// TwinCAT 3 PLC project Untitled1
// ProgramVersion: 3.1.4023.0
// libraries:
//   Tc2_SerialCom, * (Beckhoff Automation GmbH)
//   Tc2_Standard, * (Beckhoff Automation GmbH)
//   Tc2_System, * (Beckhoff Automation GmbH)
//   Tc2_Utilities, * (Beckhoff Automation GmbH)
//   Tc3_Database, * (Beckhoff Automation GmbH)
//   Tc3_IotBase, * (Beckhoff Automation GmbH)
//   Tc3_Module, * (Beckhoff Automation GmbH)
// project tree:
//   DUTs/ ST_SelectStructData.TcDUT, ST_SelectStructIMU.TcDUT
//   GVLs/ GVL.TcGVL
//   / PlcTask_Background.TcTTO, PlcTask_Buffer.TcTTO, PlcTask_Send.TcTTO, PlcTask_Read.TcTTO, PlcTask_Vacuum.TcTTO (not stored)
//   POUs/ Background_FatigueCam.TcPOU, Background_GPS.TcPOU, Background_IMU.TcPOU, Background_Time.TcPOU (not stored), Buffer_Data.TcPOU, Buffer_IMU.TcPOU, FB_FatigueCam_Receive.TcPOU (not stored), Get_Data.TcPOU, Get_IMU.TcPOU, Main_Background.TcPOU, Main_Read.TcPOU, Main_SendIMU.TcPOU, Main_Send.TcPOU, Main_Vacuum.TcPOU, Read_IMU.TcPOU, Read_Pressure.TcPOU, Read_Payload.TcPOU, Main_Buffer.TcPOU, Main_SendData.TcPOU, Read_FatigueCam.TcPOU, Read_GPS.TcPOU, Read_ID.TcPOU, Save_Data.TcPOU, Save_IMU.TcPOU, Send_Data.TcPOU, Send_IMU.TcPOU, Vacuum_Buffer_Data.TcPOU, Vacuum_Buffer_Data_2.TcPOU (not stored), Vacuum_Buffer_IMU.TcPOU, Vacuum_Buffer_IMU_2.TcPOU, Vacuum_Data.TcPOU, Vacuum_IMU.TcPOU
// real-time tasks:
//   TASK PlcTask_Buffer: cycle T#2333.1us, priority 20, ADS port 351
//   TASK PlcTask_Read: cycle T#999.9us, priority 19, ADS port 350
//   TASK PlcTask_Send: cycle T#4332.9us, priority 21, ADS port 352
//   TASK PlcTask_Background: cycle T#333.3us, priority 18, ADS port 349
//   TASK PlcTask_Vacuum: cycle T#333.3us, priority 16, ADS port 348
// I/O:
//   DEVICE Device 1 (EtherCAT) (disabled), AmsNetId 5.95.29.222.2.1
//     Term 1 (EK1200) [EK1200-5000 EtherCAT Power supply (2A E-Bus)]
//       Term 2 (EL9221-5000) [EL9221-5000 Overcurrent protection 24V DC, 1Ch., max. 10A, adjustable]
//       Term 3 (EL9011) [EL9011 End Terminal]
//   DEVICE Device 4 (EtherCAT) (disabled), AmsNetId 5.95.29.222.5.1
//     Term 4 (EK1101) [EK1101 EtherCAT Coupler (2A E-Bus, ID switch)]
//       Term 5 (EL9221-5000) [EL9221-5000 Overcurrent protection 24V DC, 1Ch., max. 10A, adjustable]
//       Term 6 (EL3052) [EL3052 2Ch. Ana. Input 4-20mA]
//       Term 7 (EL3061) [EL3061 1Ch. Ana. Input 0-10V]
//       Term 8 (EL6001) [EL6001 Interface (RS232)]
//       Term 9 (EL9505) [EL9505 Power supply terminal 5V]
//       Term 13 (EL9011) [EL9011 End Terminal]
//     Term 10 (EK1101) [EK1101 EtherCAT Coupler (2A E-Bus, ID switch)]
//       Term 11 (EL9221-5000) [EL9221-5000 Overcurrent protection 24V DC, 1Ch., max. 10A, adjustable]
//       Term 12 (EL3052) [EL3052 2Ch. Ana. Input 4-20mA]
//       Term 13 (EL3061) [EL3061 1Ch. Ana. Input 0-10V]
//       Term 14 (EL6001) [EL6001 Interface (RS232)]
//       Term 15 (EL9505) [EL9505 Power supply terminal 5V]
//       Term 14 (EL9011) [EL9011 End Terminal]
//   DEVICE Device 3 (COM Port) (disabled)
// variable links:
//   Untitled1/Untitled1 Instance <-> Device 4 (EtherCAT)/Term 10 (EK1101)
//     PlcTask_Read Inputs/GVL.Rear_Trailer_State <-> InfoData/State
//     PlcTask_Read Inputs/Read_ID.Trailer_ID_Rear <-> ID/ID
//   Untitled1/Untitled1 Instance <-> Device 4 (EtherCAT)/Term 10 (EK1101)/Term 12 (EL3052)
//     PlcTask_Read Inputs/Read_Pressure.EL3052_Rear_Bit <-> AI Standard Channel 1/Value
//   Untitled1/Untitled1 Instance <-> Device 4 (EtherCAT)/Term 10 (EK1101)/Term 13 (EL3061)
//     PlcTask_Read Inputs/Read_Payload.EL3061_Rear_Bit <-> AI Standard/Value
//   Untitled1/Untitled1 Instance <-> Device 4 (EtherCAT)/Term 10 (EK1101)/Term 14 (EL6001)
//     PlcTask_Send Inputs/Background_IMU.stIn_EL6001_Rear/D[{0..21}] <-> COM Inputs/Data In {0..21}  (22 links)
//     PlcTask_Send Inputs/Background_IMU.stIn_EL6001_Rear/Status <-> COM Inputs/Status
//     PlcTask_Send Outputs/Background_IMU.stOut_EL6001_Rear/Ctrl <-> COM Outputs/Ctrl
//     PlcTask_Send Outputs/Background_IMU.stOut_EL6001_Rear/D[{0..21}] <-> COM Outputs/Data Out {0..21}  (22 links)
//   Untitled1/Untitled1 Instance <-> Device 4 (EtherCAT)/Term 4 (EK1101)
//     PlcTask_Read Inputs/GVL.Lead_Trailer_State <-> InfoData/State
//     PlcTask_Read Inputs/Read_ID.Trailer_ID_Lead <-> ID/ID
//   Untitled1/Untitled1 Instance <-> Device 4 (EtherCAT)/Term 4 (EK1101)/Term 6 (EL3052)
//     PlcTask_Read Inputs/Read_Pressure.EL3052_Lead_Bit <-> AI Standard Channel 1/Value
//   Untitled1/Untitled1 Instance <-> Device 4 (EtherCAT)/Term 4 (EK1101)/Term 7 (EL3061)
//     PlcTask_Read Inputs/Read_Payload.EL3061_Lead_Bit <-> AI Standard/Value
//   Untitled1/Untitled1 Instance <-> Device 4 (EtherCAT)/Term 4 (EK1101)/Term 8 (EL6001)
//     PlcTask_Send Inputs/Background_IMU.stIn_EL6001_Lead/D[{0..21}] <-> COM Inputs/Data In {0..21}  (22 links)
//     PlcTask_Send Inputs/Background_IMU.stIn_EL6001_Lead/Status <-> COM Inputs/Status
//     PlcTask_Send Outputs/Background_IMU.stOut_EL6001_Lead/Ctrl <-> COM Outputs/Ctrl
//     PlcTask_Send Outputs/Background_IMU.stOut_EL6001_Lead/D[{0..21}] <-> COM Outputs/Data Out {0..21}  (22 links)

CONFIGURATION Untitled1
    RESOURCE PLC ON TwinCAT3
        TASK PlcTask_Background(INTERVAL := ?, PRIORITY := 18);
        TASK PlcTask_Buffer(INTERVAL := T#2333.1us, PRIORITY := 20);
        TASK PlcTask_Send(INTERVAL := T#97323.6us, PRIORITY := 21);
        TASK PlcTask_Read(INTERVAL := T#999.9us, PRIORITY := 19);
        PROGRAM Main_Background WITH PlcTask_Background : Main_Background;
        PROGRAM Main_Buffer WITH PlcTask_Buffer : Main_Buffer;
        PROGRAM Main_Send WITH PlcTask_Send : Main_Send;
        PROGRAM Main_Read WITH PlcTask_Read : Main_Read;
    END_RESOURCE
END_CONFIGURATION

// ---- DUTs/ST_SelectStructData.TcDUT
TYPE ST_SelectStructData :
STRUCT
	TimeStr			: DATE_AND_TIME;	
	Trailer_ID		: UINT;
	Lat				: LREAL;
	Lon				: LREAL;
	Speed			: LREAL;
	Overspeed		: BOOL;
	Payload_EMA		: LREAL;
	Payload_Raw		: LREAL;
	Overload		: BOOL;
	Pressure_Cyl	: LREAL;
	Pressure_Val	: LREAL;
	Strain_Left		: LREAL;
	Strain_Right	: LREAL;
	EventCode		: UINT;
	Cycle_Duration	: UDINT;
	Hyd_Efficiency	: LREAL;
END_STRUCT
END_TYPE

// ---- DUTs/ST_SelectStructIMU.TcDUT
TYPE ST_SelectStructIMU :
STRUCT
	TimeStr			: DATE_AND_TIME;
	Millis			: UINT;	
	Trailer_ID		: UINT;
	RoadSec			: UINT;
	AccX			: LREAL;
	AccY			: LREAL;
	AccZ			: LREAL;
	Pitch			: LREAL;
	Roll			: LREAL;
END_STRUCT
END_TYPE

// ---- GVLs/GVL.TcGVL
{attribute 'qualified_only'}
VAR_GLOBAL
	Lead_Trailer_State AT %I*	: UINT;
	Rear_Trailer_State AT %I*	: UINT;
END_VAR

// ---- POUs/Main_Background.TcPOU
PROGRAM Main_Background
VAR
END_VAR

(* execute background processes *)
Background_Time();
//Background_IMU();
//Background_FatigueCam();
Background_GPS();

END_PROGRAM

// ---- POUs/Background_GPS.TcPOU
PROGRAM Background_GPS

VAR
	RxBuffer	:ComBuffer;
	TxBuffer	:ComBuffer;
	
	fbLineCtrlAds	: SerialLineControlADS;
	bAdsError		: BOOL;
	nAdsErrorID		: UDINT;
	bConnect		: BOOL := TRUE;
	sNetID			: T_amsNetId;
	stSerialCfg		: ComSerialConfig;
	Port			: BOOL;
END_VAR

stSerialCfg.Baudrate := 4800;
stSerialCfg.ComPort := 3;
stSerialCfg.DataBits := 8;
stSerialCfg.Parity := PARITY_NONE;
stSerialCfg.StopBits := STOPBITS_ONE;

fbLineCtrlAds(
	Connect 	:= bConnect,
	SerialCfg	:= stSerialCfg,
	NetId		:= sNetId,
	Timeout		:= T#5s,
	TxBuffer	:= TxBuffer,
	RxBuffer	:= RxBuffer,
	Busy		:= ,
	Error		=> bAdsError,
	ErrorID		=> nAdsErrorID,
	PortOpened	=> Port
);

END_PROGRAM

// ---- POUs/Main_Buffer.TcPOU
PROGRAM Main_Buffer
VAR
	
END_VAR

(* save data to database *)
//Buffer_Data();
Buffer_IMU();

END_PROGRAM

// ---- POUs/Buffer_IMU.TcPOU
PROGRAM Buffer_IMU
VAR
	pSec		: WORD;
	diff		: BOOL;
	
	TimeStr		: ARRAY [1..50] OF STRING;
	//Millis		: ARRAY [1..50] OF STRING;
	Trailer_ID_Lead	: ARRAY [1..50] OF STRING;
	//RoadSec		: ARRAY [1..50] OF STRING;
	Pitch_Lead		: ARRAY [1..50] OF STRING;
	Roll_Lead		: ARRAY [1..50] OF STRING;
	AccX_Lead		: ARRAY [1..50] OF STRING;
	AccY_Lead		: ARRAY [1..50] OF STRING;
	AccZ_Lead		: ARRAY [1..50] OF STRING;
	
	Trailer_ID_Rear	: ARRAY [1..50] OF STRING;
	//RoadSec		: ARRAY [1..50] OF STRING;
	Pitch_Rear		: ARRAY [1..50] OF STRING;
	Roll_Rear		: ARRAY [1..50] OF STRING;
	AccX_Rear		: ARRAY [1..50] OF STRING;
	AccY_Rear		: ARRAY [1..50] OF STRING;
	AccZ_Rear		: ARRAY [1..50] OF STRING;
	
	fbSqlDatabase	: FB_SQLDatabaseEvt(sNetID := '', tTimeout := T#1000S);
	fbSqlCommand	: FB_SQLCommandEvt(sNetID := '', tTimeout := T#1000S);
	fbSqlResult		: FB_SQLResultEvt(sNetID:='', tTimeout   := T#1000S); 
	sCmd			: STRING(500000);
	sCmd2			: STRING(500000);
	nState			: INT;
	nState_Switch	: INT;
	
	aReadStruct		: ST_SelectStructIMU;
	aReadStruct_2	: ST_SelectStructIMU;
	Timestamp		: DT;
	Timestamp_2		: DT; 
	
	Initialized		: BOOL := FALSE;
	Done			: BOOL;
	i				: INT;
	Pragma_Done		: BOOL;
	Counter			: ULINT;
	
	Dbid			: UDINT;
	
	bDisconnect		: BOOL;
END_VAR

(* convert to strings *)
//PrimeMover_ID		:= Read_ID.PrimeMover_ID;
TimeStr				:= Read_IMU.TimeStr;
//Millis			:= Read_IMU.Millis;
Trailer_ID_Lead		:= Read_IMU.Trailer_ID_Lead;
Pitch_Lead			:= Read_IMU.Pitch_Lead;
Roll_Lead			:= Read_IMU.Roll_Lead;
AccX_Lead			:= Read_IMU.AccX_Lead;
AccY_Lead			:= Read_IMU.AccY_Lead;
AccZ_Lead			:= Read_IMU.AccZ_Lead;

Trailer_ID_Rear		:= Read_IMU.Trailer_ID_Rear;
Pitch_Rear			:= Read_IMU.Pitch_Rear;
Roll_Rear			:= Read_IMU.Roll_Rear;
AccX_Rear			:= Read_IMU.AccX_Rear;
AccY_Rear			:= Read_IMU.AccY_Rear;
AccZ_Rear			:= Read_IMU.AccZ_Rear;

IF NOT Initialized THEN
	
	//initialization (choose which database for buffer)
	CASE nState OF
				
		0:
			(* connect to buffer_imu *)	
			IF Vacuum_Buffer_IMU.Vacuumed THEN
				
				Dbid := 2;		
				IF fbSqlDatabase.Connect(Dbid) THEN
					IF fbSqlDatabase.bError THEN
						nState := 255; 
					ELSE
						nState := nState+1;
					END_IF
				END_IF
				
			END_IF
			
			
		1:
			IF fbSqlDatabase.CreateCmd(ADR(fbSqlCommand)) THEN
				IF fbSqlDatabase.bError THEN
					nState := 255; 
				ELSE
					nState := nState+1; 
				END_IF
			END_IF
			
		2:	(* execute pragmas *)
			sCmd	:= 'PRAGMA journal_mode = WAL; PRAGMA synchronous = NORMAL; PRAGMA temp_store = MEMORY; PRAGMA mmap_size = 30000000000; PRAGMA page_size = 32768; PRAGMA locking_mode = EXCLUSIVE;';
			
			IF fbSQLCommand.Execute(ADR(sCmd), SIZEOF(sCmd)) THEN
				IF fbSQLCommand.bError THEN
					nState := 255; 
				ELSE
					nState := nState+1; 
				END_IF
			END_IF
			
		3:
			(* select oldest data from buffer_imu *)
			sCmd	:= 'SELECT * FROM `buffer_imu` ORDER BY datetime ASC LIMIT 1';
			
			IF fbSQLCommand.ExecuteDataReturn(ADR(sCmd), SIZEOF(sCmd), ADR(fbSqlResult)) THEN
				IF fbSQLCommand.bError THEN
					nState := 255; 
				ELSE
					nState := nState+1; 
				END_IF
			END_IF
			
		4:
			IF fbSqlResult.Read(0, 1, ADR(aReadStruct), SIZEOF(aReadStruct), TRUE, TRUE) THEN
				IF fbSqlResult.bError THEN
					nState := 255; 
				ELSE
					nState := nState+1; 
				END_IF
			END_IF
			
		5:
			IF fbSqlResult.Release() THEN
				IF fbSqlResult.bError THEN
					nState := 255;
				ELSE
					nState := nState+1;
				END_IF
			END_IF
			
		6:	(* execute pragma optimize *)
			sCmd	:= 'PRAGMA optimize;';
			
			IF fbSQLCommand.Execute(ADR(sCmd), SIZEOF(sCmd)) THEN
				IF fbSQLCommand.bError THEN
					nState := 255; 
				ELSE
					nState := nState+1; 
				END_IF
			END_IF
			
		7:
			(* disconnect from buffer_imu *)
			IF fbSqlDatabase.Disconnect() THEN
				IF fbSqlDatabase.bError THEN
					nState := 255;
				ELSE
					nState := nState+1;
				END_IF
			END_IF
			
		8:	
			(* connect to buffer_imu_2 *)
			IF Vacuum_Buffer_IMU_2.Vacuumed THEN
				
				Dbid := 5;	
				IF fbSqlDatabase.Connect(Dbid) THEN
					IF fbSqlDatabase.bError THEN
						nState := 255; 
					ELSE
						nState := nState+1;
					END_IF
				END_IF
				
			END_IF	
			
		9:
			IF fbSqlDatabase.CreateCmd(ADR(fbSqlCommand)) THEN
				IF fbSqlDatabase.bError THEN
					nState := 255; 
				ELSE
					nState := nState+1; 
				END_IF
			END_IF
			
		10:	(* execute pragmas *)
			sCmd	:= 'PRAGMA journal_mode = WAL; PRAGMA synchronous = NORMAL; PRAGMA temp_store = MEMORY; PRAGMA mmap_size = 30000000000; PRAGMA page_size = 32768; PRAGMA locking_mode = EXCLUSIVE;';
			
			IF fbSQLCommand.Execute(ADR(sCmd), SIZEOF(sCmd)) THEN
				IF fbSQLCommand.bError THEN
					nState := 255; 
				ELSE
					nState := nState+1; 
				END_IF
			END_IF
			
		11:
			(* select oldest data from buffer_imu *)
			sCmd	:= 'SELECT * FROM `buffer_imu` ORDER BY datetime ASC LIMIT 1';
			
			IF fbSQLCommand.ExecuteDataReturn(ADR(sCmd), SIZEOF(sCmd), ADR(fbSqlResult)) THEN
				IF fbSQLCommand.bError THEN
					nState := 255; 
				ELSE
					nState := nState+1; 
				END_IF
			END_IF
			
		12:
			IF fbSqlResult.Read(0, 1, ADR(aReadStruct_2), SIZEOF(aReadStruct_2), TRUE, TRUE) THEN
				IF fbSqlResult.bError THEN
					nState := 255; 
				ELSE
					nState := nState+1; 
				END_IF
			END_IF
			
		13:
			IF fbSqlResult.Release() THEN
				IF fbSqlResult.bError THEN
					nState := 255;
				ELSE
					nState := nState+1;
				END_IF
			END_IF
			
		14:	(* execute pragma optimize *)
			sCmd	:= 'PRAGMA optimize;';
			
			IF fbSQLCommand.Execute(ADR(sCmd), SIZEOF(sCmd)) THEN
				IF fbSQLCommand.bError THEN
					nState := 255; 
				ELSE
					nState := nState+1; 
				END_IF
			END_IF
			
		15:
			(* disconnect from buffer_imu_2 *)
			IF bDisconnect := fbSqlDatabase.Disconnect() THEN
				IF fbSqlDatabase.bError THEN
					nState := 255;
				ELSE
					nState := nState+1;
				END_IF
			END_IF
			
		16:
			// compare oldest data
			aReadStruct.datetime 	:= REPLACE(aReadStruct.datetime, '-', 1, 11);
			aReadStruct_2.datetime 	:= REPLACE(aReadStruct_2.datetime, '-', 1, 11);
			
			Timestamp	:= SYSTEMTIME_TO_DT(STRING_TO_SYSTEMTIME(aReadStruct.datetime));
			Timestamp_2	:= SYSTEMTIME_TO_DT(STRING_TO_SYSTEMTIME(aReadStruct_2.datetime));

			IF Timestamp = DT#1970-1-1-00:00:00 THEN
				Dbid := 2;
			ELSIF Timestamp_2 = DT#1970-1-1-00:00:00 THEN
				Dbid := 5;
			ELSIF Timestamp > Timestamp_2 THEN
				Dbid := 2;
			ELSE
				Dbid := 5;
			END_IF
			
			Initialized := TRUE;
			nState		:= 0;
			
		255:
			nState := 0;
			
	END_CASE

ELSE	
	
	(* save data to buffer every second *)
	IF diff:= Background_Time.cSec <> pSec THEN
		
		//database switching
		IF Get_IMU.Switch AND Counter >= 750 THEN
			
			CASE nState_Switch OF
				
				0:	(* execute pragma optimize *)
					sCmd	:= 'PRAGMA optimize;';
					
					IF fbSQLCommand.Execute(ADR(sCmd), SIZEOF(sCmd)) THEN
						IF fbSQLCommand.bError THEN
							nState_Switch := 255; 
						ELSE
							nState_Switch := nState_Switch+1; 
						END_IF
					END_IF
				
				1:
					IF fbSqlDatabase.bConnected THEN
						fbSqlDatabase.Disconnect();
					ELSE
						IF Dbid = 2 THEN
							Dbid := 5;
						ELSE
							Dbid := 2;
						END_IF
						Counter			:= 0;
						nState_Switch 	:= 0;
						Pragma_Done		:= FALSE;
					END_IF
					
				255:
					nState_Switch := 0;
					
			END_CASE
		
		ELSE
			
			IF Done THEN
				Done	:= FALSE;
				IF fbSqlDatabase.bConnected THEN
					nState 	:= 1;
				ELSE
					nState 	:= 0;
				END_IF	
			END_IF
			
			CASE nState OF	
				0:	
					IF fbSqlDatabase.Connect(Dbid) THEN
						IF fbSqlDatabase.bError THEN
							nState := 255;
						ELSE
							nState := nState + 1; 
						END_IF
					END_IF
				
				1:
					IF fbSqlDatabase.CreateCmd(ADR(fbSqlCommand)) THEN
						IF fbSqlDatabase.bError THEN
							nState := 255; 
						ELSE
							nState := nState+1; 
						END_IF
					END_IF
					
				2:	(* execute pragmas *)
					IF NOT Pragma_Done THEN
						sCmd	:= 'PRAGMA journal_mode = WAL; PRAGMA synchronous = NORMAL; PRAGMA temp_store = MEMORY; PRAGMA mmap_size = 30000000000; PRAGMA page_size = 32768; PRAGMA locking_mode = EXCLUSIVE;';
					
						IF fbSQLCommand.Execute(ADR(sCmd), SIZEOF(sCmd)) THEN
							IF fbSQLCommand.bError THEN
								nState := 255; 
							ELSE
								nState 		:= nState+1; 
								Pragma_Done := TRUE;
							END_IF
						END_IF
					
					ELSE
						nState 		:= nState+1;
 
					END_IF
					
				3:	
					(* build query *)	
					sCmd:= 'INSERT INTO buffer_imu (datetime,trailer_id_lead,trailer_id_rear,pitch_lead,roll_lead,ax_lead,ay_lead,az_lead,pitch_rear,roll_rear,ax_rear,ay_rear,az_rear) VALUES ';
					
					FOR i := 1 TO 50 BY 1 DO
						sCmd2:= CONCAT('($'', TimeStr[i]);
						sCmd2:= CONCAT(sCmd2, '$',');
						sCmd2:= CONCAT(sCmd2, Trailer_ID_Lead[i]);
						sCmd2:= CONCAT(sCmd2, ',');
						sCmd2:= CONCAT(sCmd2, Trailer_ID_Rear[i]);
						sCmd2:= CONCAT(sCmd2, ',');
						sCmd2:= CONCAT(sCmd2, Pitch_Lead[i]);
						sCmd2:= CONCAT(sCmd2, ',');
						sCmd2:= CONCAT(sCmd2, Roll_Lead[i]);
						sCmd2:= CONCAT(sCmd2, ',');
						sCmd2:= CONCAT(sCmd2, AccX_Lead[i]);
						sCmd2:= CONCAT(sCmd2, ',');
						sCmd2:= CONCAT(sCmd2, AccY_Lead[i]);
						sCmd2:= CONCAT(sCmd2, ',');
						sCmd2:= CONCAT(sCmd2, AccZ_Lead[i]);
						sCmd2:= CONCAT(sCmd2, ',');
						sCmd2:= CONCAT(sCmd2, Pitch_Rear[i]);
						sCmd2:= CONCAT(sCmd2, ',');
						sCmd2:= CONCAT(sCmd2, Roll_Rear[i]);
						sCmd2:= CONCAT(sCmd2, ',');
						sCmd2:= CONCAT(sCmd2, AccX_Rear[i]);
						sCmd2:= CONCAT(sCmd2, ',');
						sCmd2:= CONCAT(sCmd2, AccY_Rear[i]);
						sCmd2:= CONCAT(sCmd2, ',');
						sCmd2:= CONCAT(sCmd2, AccZ_Rear[i]);
						
						IF i = 50 THEN
							sCmd2:= CONCAT(sCmd2, ')');
						ELSE	
							sCmd2:= CONCAT(sCmd2, '),');
						END_IF
						
						CONCAT2(ADR(sCmd), ADR(sCmd2), ADR(sCmd), SIZEOF(sCmd));
					END_FOR
					
					
					IF fbSQLCommand.Execute(ADR(sCmd), SIZEOF(sCmd)) THEN
						IF fbSQLCommand.bError THEN
							nState := 255; 
						ELSE
							nState := nState+1; 
							pSec := Background_Time.cSec;
							
						END_IF
					END_IF
					
				4: 
					Counter := Counter + 50;
					Done	:= TRUE;
						
				255:
					nState := 0;
					
			END_CASE	
			
		END_IF
	END_IF
END_IF

END_PROGRAM

// ---- POUs/Read_IMU.TcPOU
PROGRAM Read_IMU
VAR
	
	cSec		: WORD;
	pSec		: WORD;
	i			: INT := 1;
	j			: INT;
	
	TimeStr				: ARRAY [1..50] OF STRING;
	Trailer_ID_Lead		: ARRAY [1..50] OF STRING;
	//RoadSec			: ARRAY [1..50] OF UINT;
	Pitch_Lead			: ARRAY [1..50] OF STRING;
	Roll_Lead			: ARRAY [1..50] OF STRING;
	AccX_Lead			: ARRAY [1..50] OF STRING;
	AccY_Lead			: ARRAY [1..50] OF STRING;
	AccZ_Lead			: ARRAY [1..50] OF STRING;
	
	Trailer_ID_Rear	: ARRAY [1..50] OF STRING;
	//RoadSec		: ARRAY [1..50] OF UINT;
	Pitch_Rear		: ARRAY [1..50] OF STRING;
	Roll_Rear		: ARRAY [1..50] OF STRING;
	AccX_Rear		: ARRAY [1..50] OF STRING;
	AccY_Rear		: ARRAY [1..50] OF STRING;
	AccZ_Rear		: ARRAY [1..50] OF STRING;
	
	cDiv	: UINT;
	pDiv	: UINT;

END_VAR

cDiv	:= Background_Time.cMil / 20; 
	
IF pSec <> Background_Time.cSec THEN 
	j := i;
	i := 1;
	pSec := Background_Time.cSec;
END_IF
	
IF pDiv <> cDiv THEN
	
	TimeStr[i]				:= REPLACE(Background_Time.TimeStr, ' ', 1, 11);
	
	IF GVL.Lead_Trailer_State = 8 OR GVL.Lead_Trailer_State = 17416 THEN
		Trailer_ID_Lead[i]		:= UINT_TO_STRING(Read_ID.Trailer_ID_Lead);
		//RoadSec[i]			:= Background_IMU.RoadSec;
		Pitch_Lead[i]			:= REAL_TO_STRING(Background_IMU.Pitch_Lead);
		Roll_Lead[i]			:= REAL_TO_STRING(Background_IMU.Roll_Lead);
		AccX_Lead[i]			:= REAL_TO_STRING(Background_IMU.AccX_Lead);
		AccY_Lead[i]			:= REAL_TO_STRING(Background_IMU.AccY_Lead);
		AccZ_Lead[i]			:= REAL_TO_STRING(Background_IMU.AccZ_Lead);
	ELSE
		Trailer_ID_Lead[i]		:= '99';
		//RoadSec[i]			:= Background_IMU.RoadSec;
		Pitch_Lead[i]			:= '0';
		Roll_Lead[i]			:= '0';
		AccX_Lead[i]			:= '0';
		AccY_Lead[i]			:= '0';
		AccZ_Lead[i]			:= '0';
	END_IF
	
	IF GVL.Rear_Trailer_State = 8 THEN
		Trailer_ID_Rear[i]		:= UINT_TO_STRING(Read_ID.Trailer_ID_Rear);
		//RoadSec[i]			:= Background_IMU.RoadSec;
		Pitch_Rear[i]			:= REAL_TO_STRING(Background_IMU.Pitch_Rear);
		Roll_Rear[i]			:= REAL_TO_STRING(Background_IMU.Roll_Rear);
		AccX_Rear[i]			:= REAL_TO_STRING(Background_IMU.AccX_Rear);
		AccY_Rear[i]			:= REAL_TO_STRING(Background_IMU.AccY_Rear);
		AccZ_Rear[i]			:= REAL_TO_STRING(Background_IMU.AccZ_Rear);
	ELSE
		Trailer_ID_Rear[i]		:= '99';
		//RoadSec[i]			:= Background_IMU.RoadSec;
		Pitch_Rear[i]			:= '0';
		Roll_Rear[i]			:= '0';
		AccX_Rear[i]			:= '0';
		AccY_Rear[i]			:= '0';
		AccZ_Rear[i]			:= '0';
	END_IF
	
	pDiv := cDiv;
	i := i+1;
	
END_IF;

END_PROGRAM

// ---- POUs/Read_ID.TcPOU
PROGRAM Read_ID
VAR
	PrimeMover_ID			: STRING := '99';
	Trailer_ID_Lead AT %I*	: UINT;
	Trailer_ID_Rear AT %I*	: UINT;
END_VAR

;

END_PROGRAM

// ---- POUs/Background_IMU.TcPOU
PROGRAM Background_IMU
VAR
	(* background communication with the EL6001 terminal *)
	fbEL6001Ctrl		: SerialLineControl;
	
	bEL6001CtrlError_Lead	: BOOL;
	eEL6001CtrlErrorID_Lead	: ComError_t;
	bEL6001CtrlError_Rear	: BOOL;
	eEL6001CtrlErrorID_Rear	: ComError_t;
	
	(* 	I/O variables for a EL6001 terminal*)
	stIn_EL6001_Lead AT %I*		: EL6inData22B;	(* linked to the EL6001 in the TwinCAT System Manager *)
	stOut_EL6001_Lead AT %Q*	: EL6outData22B;(* linked to the EL6001 in the TwinCAT System Manager *)
	RxBuffer_Lead				: ComBuffer;
	TxBuffer_Lead				: ComBuffer;
	
	stIn_EL6001_Rear AT %I*		: EL6inData22B;	(* linked to the EL6001 in the TwinCAT System Manager *)
	stOut_EL6001_Rear AT %Q*	: EL6outData22B;(* linked to the EL6001 in the TwinCAT System Manager *)
	RxBuffer_Rear				: ComBuffer;
	TxBuffer_Rear				: ComBuffer;
	
	fbReceive		: ReceiveData;
	fbClearCom		: ClearComBuffer;
	Prefix			: UINT := 16#2F77;
	nReceiveCounter	: UDINT := 1;
	
	bReceiveBusy_Lead		: BOOL;
	bReceiveError_Lead		: BOOL;
	eReceiveErrorID_Lead	: ComError_t;
	bReceiveTimeout_Lead	: BOOL;
	bDataReceived_Lead		: BOOL;
	
	bReceiveBusy_Rear		: BOOL;
	bReceiveError_Rear		: BOOL;
	eReceiveErrorID_Rear	: ComError_t;
	bReceiveTimeout_Rear	: BOOL;
	bDataReceived_Rear		: BOOL;
	
	Data_Lead		: ARRAY [1..6] OF ULINT;
	DataStr_Lead	: ARRAY [1..6] OF STRING;
	Data_Rear		: ARRAY [1..6] OF ULINT;
	DataStr_Rear	: ARRAY [1..6] OF STRING;
	
	Counter_Lead	: UINT := 0;
	Total_Lead		: UINT;
	
	Counter_Rear	: UINT := 0;
	Total_Rear		: UINT;
	
	//RoadSec	: UINT := 0;
	Pitch_Lead	: REAL;
	Roll_Lead	: REAL;
	AccX_Lead	: REAL; //along pitch axis, perpendicular to driving direction 
	AccY_Lead	: REAL;	//along roll axis, parallel to driving direction
	AccZ_Lead	: REAL;
	
	Pitch_Rear	: REAL;
	Roll_Rear	: REAL;
	AccX_Rear	: REAL; //along pitch axis, perpendicular to driving direction 
	AccY_Rear	: REAL;	//along roll axis, parallel to driving direction
	AccZ_Rear	: REAL;
	
	pSec		: WORD;
END_VAR

(* background communication with the EL6001 terminal *)
fbEL6001Ctrl(
	Mode:= SERIALLINEMODE_EL6_22B, 
	pComIn:= ADR(stIn_EL6001_Lead), 
	pComOut:= ADR(stOut_EL6001_Lead), 
	SizeComIn:= SIZEOF(stIn_EL6001_Lead), 
	Error=> , 
	ErrorID=> , 
	TxBuffer:= TxBuffer_Lead, 
	RxBuffer:= RxBuffer_Lead );
IF fbEL6001Ctrl.Error THEN
	bEL6001CtrlError_Lead := TRUE;
	eEL6001CtrlErrorID_Lead := fbEL6001Ctrl.ErrorID;
END_IF

fbEL6001Ctrl(
	Mode:= SERIALLINEMODE_EL6_22B, 
	pComIn:= ADR(stIn_EL6001_Rear), 
	pComOut:= ADR(stOut_EL6001_Rear), 
	SizeComIn:= SIZEOF(stIn_EL6001_Rear), 
	Error=> , 
	ErrorID=> , 
	TxBuffer:= TxBuffer_Rear, 
	RxBuffer:= RxBuffer_Rear );
IF fbEL6001Ctrl.Error THEN
	bEL6001CtrlError_Rear := TRUE;
	eEL6001CtrlErrorID_Rear := fbEL6001Ctrl.ErrorID;
END_IF

(* read data from imu *)
fbReceive( 
	RxBuffer := RxBuffer_Lead,
	pPrefix := ADR(Prefix),
	LenPrefix := 2,
	pReceiveData := ADR(Data_Lead),
	SizeReceiveData	:= 48,
	Timeout:= T#1S,
	Busy => bReceiveBusy_Lead,
	Error => ,
	DataReceived => bDataReceived_Lead,
	RxTimeout=> bReceiveTimeout_Lead
);

IF fbReceive.Error <> COMERROR_NOERROR THEN
	eReceiveErrorID_Lead := fbReceive.Error;
	
END_IF

fbReceive( 
	RxBuffer := RxBuffer_Rear,
	pPrefix := ADR(Prefix),
	LenPrefix := 2,
	pReceiveData := ADR(Data_Rear),
	SizeReceiveData	:= 48,
	Timeout:= T#1S,
	Busy => bReceiveBusy_Rear,
	Error => ,
	DataReceived => bDataReceived_Rear,
	RxTimeout=> bReceiveTimeout_Rear 
);

IF fbReceive.Error <> COMERROR_NOERROR THEN
	eReceiveErrorID_Rear := fbReceive.Error;
	
END_IF

IF bDataReceived_Lead THEN
	fbClearCom(Buffer := RxBuffer_Lead); //clear rx buffer
	
	(* parse data *)
	DataStr_Lead[1]	:= LWORD_TO_HEXSTR(in := Data_Lead[1], iPrecision := 16, bLoCase := FALSE);
	DataStr_Lead[2]	:= LWORD_TO_HEXSTR(in := Data_Lead[2], iPrecision := 16, bLoCase := FALSE);
	DataStr_Lead[3]	:= LWORD_TO_HEXSTR(in := Data_Lead[3], iPrecision := 16, bLoCase := FALSE);
	DataStr_Lead[4]	:= LWORD_TO_HEXSTR(in := Data_Lead[4], iPrecision := 16, bLoCase := FALSE);
	
	(* parse pitch *)
	Pitch_Lead	:= (100 * STRING_TO_REAL(MID(DataStr_Lead[1], 1, 8))) + STRING_TO_REAL(MID(DataStr_Lead[1], 2, 5)) +  (0.01 * STRING_TO_REAL(MID(DataStr_Lead[1], 2, 3)));
	IF MID(DataStr_Lead[1], 1, 7) = '1' THEN
		Pitch_Lead	:= Pitch_Lead * (-1);
		
	END_IF
		
	(* parse roll *)
	Roll_Lead	:= (100 * STRING_TO_REAL(MID(DataStr_Lead[1], 1, 2))) + STRING_TO_REAL(MID(DataStr_Lead[2], 2, 15)) +  (0.01 * STRING_TO_REAL(MID(DataStr_Lead[2], 2, 13)));
	IF MID(DataStr_Lead[1], 1, 1) = '1' THEN
		Roll_Lead	:= Roll_Lead * (-1);
		
	END_IF
		
	(* parse accx *)
	IF MID(DataStr_Lead[2], 1, 6) = 'A' THEN
		AccX_Lead	:= 10;
		
	ELSIF MID(DataStr_Lead[2], 1, 6) = 'B' THEN
		AccX_Lead	:= 11;
		
	ELSIF MID(DataStr_Lead[2], 1, 6) = 'C' THEN
		AccX_Lead	:= 12;
		
	ELSIF MID(DataStr_Lead[2], 1, 6) = 'D' THEN
		AccX_Lead	:= 13;
		
	ELSIF MID(DataStr_Lead[2], 1, 6) = 'E' THEN
		AccX_Lead	:= 14;
	
	ELSIF MID(DataStr_Lead[2], 1, 6) = 'F' THEN
		AccX_Lead	:= 15;
		
	ELSE
		AccX_Lead	:= STRING_TO_REAL(MID(DataStr_Lead[2], 1, 6));	
	
	END_IF
	
	AccX_Lead	:=  AccX_Lead + (0.01 * STRING_TO_REAL(MID(DataStr_Lead[2], 2, 3))) +  (0.0001 * STRING_TO_REAL(MID(DataStr_Lead[2], 2, 1)));
	IF MID(DataStr_Lead[2], 1, 5) = '1' THEN
		AccX_Lead	:= AccX_Lead * (-1);
		
	END_IF
	
	(* parse accy *)
	IF MID(DataStr_Lead[3], 1, 16) = 'A' THEN
		AccY_Lead	:= 10;
		
	ELSIF MID(DataStr_Lead[3], 1, 16) = 'B' THEN
		AccY_Lead	:= 11;
		
	ELSIF MID(DataStr_Lead[3], 1, 16) = 'C' THEN
		AccY_Lead	:= 12;
		
	ELSIF MID(DataStr_Lead[3], 1, 16) = 'D' THEN
		AccY_Lead	:= 13;
		
	ELSIF MID(DataStr_Lead[3], 1, 16) = 'E' THEN
		AccY_Lead	:= 14;
	
	ELSIF MID(DataStr_Lead[3], 1, 16) = 'F' THEN
		AccY_Lead	:= 15;
		
	ELSE
		AccY_Lead	:= STRING_TO_REAL(MID(DataStr_Lead[3], 1, 16));	
	
	END_IF
	
	AccY_Lead	:=  AccY_Lead + (0.01 * STRING_TO_REAL(MID(DataStr_Lead[3], 2, 13))) +  (0.0001 * STRING_TO_REAL(MID(DataStr_Lead[3], 2, 11)));
	IF MID(DataStr_Lead[3], 1, 15) = '1' THEN
		AccY_Lead	:= AccY_Lead * (-1);
		
	END_IF
	
	(* parse accz *)
	IF MID(DataStr_Lead[3], 1, 10) = 'A' THEN
		AccZ_Lead	:= 10;
		
	ELSIF MID(DataStr_Lead[3], 1, 10) = 'B' THEN
		AccZ_Lead	:= 11;
		
	ELSIF MID(DataStr_Lead[3], 1, 10) = 'C' THEN
		AccZ_Lead	:= 12;
		
	ELSIF MID(DataStr_Lead[3], 1, 10) = 'D' THEN
		AccZ_Lead	:= 13;
		
	ELSIF MID(DataStr_Lead[3], 1, 10) = 'E' THEN
		AccZ_Lead	:= 14;
	
	ELSIF MID(DataStr_Lead[3], 1, 10) = 'F' THEN
		AccZ_Lead	:= 15;
		
	ELSE
		AccZ_Lead	:= STRING_TO_REAL(MID(DataStr_Lead[3], 1, 10));	
	
	END_IF
	
	AccZ_Lead	:=  AccZ_Lead + (0.01 * STRING_TO_REAL(MID(DataStr_Lead[3], 2, 7))) +  (0.0001 * STRING_TO_REAL(MID(DataStr_Lead[3], 2, 5)));
	IF MID(DataStr_Lead[3], 1, 9) = '1' THEN
		AccZ_Lead	:= AccZ_Lead * (-1);
		
	END_IF
	
	(* detect road section *)
	//algorithm for road section detection
	
	Counter_Lead			:= Counter_Lead + 1;	
	
END_IF

IF bDataReceived_Rear THEN
	fbClearCom(Buffer := RxBuffer_Rear); //clear rx buffer
	
	(* parse data *)
	DataStr_Rear[1]	:= LWORD_TO_HEXSTR(in := Data_Rear[1], iPrecision := 16, bLoCase := FALSE);
	DataStr_Rear[2]	:= LWORD_TO_HEXSTR(in := Data_Rear[2], iPrecision := 16, bLoCase := FALSE);
	DataStr_Rear[3]	:= LWORD_TO_HEXSTR(in := Data_Rear[3], iPrecision := 16, bLoCase := FALSE);
	DataStr_Rear[4]	:= LWORD_TO_HEXSTR(in := Data_Rear[4], iPrecision := 16, bLoCase := FALSE);
	
	(* parse pitch *)
	Pitch_Rear	:= (100 * STRING_TO_REAL(MID(DataStr_Rear[1], 1, 8))) + STRING_TO_REAL(MID(DataStr_Rear[1], 2, 5)) +  (0.01 * STRING_TO_REAL(MID(DataStr_Rear[1], 2, 3)));
	IF MID(DataStr_Rear[1], 1, 7) = '1' THEN
		Pitch_Rear	:= Pitch_Rear * (-1);
		
	END_IF
		
	(* parse roll *)
	Roll_Rear	:= (100 * STRING_TO_REAL(MID(DataStr_Rear[1], 1, 2))) + STRING_TO_REAL(MID(DataStr_Rear[2], 2, 15)) +  (0.01 * STRING_TO_REAL(MID(DataStr_Rear[2], 2, 13)));
	IF MID(DataStr_Rear[1], 1, 1) = '1' THEN
		Roll_Rear	:= Roll_Rear * (-1);
		
	END_IF
		
	(* parse accx *)
	IF MID(DataStr_Rear[2], 1, 6) = 'A' THEN
		AccX_Rear	:= 10;
		
	ELSIF MID(DataStr_Rear[2], 1, 6) = 'B' THEN
		AccX_Rear	:= 11;
		
	ELSIF MID(DataStr_Rear[2], 1, 6) = 'C' THEN
		AccX_Rear	:= 12;
		
	ELSIF MID(DataStr_Rear[2], 1, 6) = 'D' THEN
		AccX_Rear	:= 13;
		
	ELSIF MID(DataStr_Rear[2], 1, 6) = 'E' THEN
		AccX_Rear	:= 14;
	
	ELSIF MID(DataStr_Rear[2], 1, 6) = 'F' THEN
		AccX_Rear	:= 15;
		
	ELSE
		AccX_Rear	:= STRING_TO_REAL(MID(DataStr_Rear[2], 1, 6));	
	
	END_IF
	
	AccX_Rear	:=  AccX_Rear + (0.01 * STRING_TO_REAL(MID(DataStr_Rear[2], 2, 3))) +  (0.0001 * STRING_TO_REAL(MID(DataStr_Rear[2], 2, 1)));
	IF MID(DataStr_Rear[2], 1, 5) = '1' THEN
		AccX_Rear	:= AccX_Rear * (-1);
		
	END_IF
	
	(* parse accy *)
	IF MID(DataStr_Rear[3], 1, 16) = 'A' THEN
		AccY_Rear	:= 10;
		
	ELSIF MID(DataStr_Rear[3], 1, 16) = 'B' THEN
		AccY_Rear	:= 11;
		
	ELSIF MID(DataStr_Rear[3], 1, 16) = 'C' THEN
		AccY_Rear	:= 12;
		
	ELSIF MID(DataStr_Rear[3], 1, 16) = 'D' THEN
		AccY_Rear	:= 13;
		
	ELSIF MID(DataStr_Rear[3], 1, 16) = 'E' THEN
		AccY_Rear	:= 14;
	
	ELSIF MID(DataStr_Rear[3], 1, 16) = 'F' THEN
		AccY_Rear	:= 15;
		
	ELSE
		AccY_Rear	:= STRING_TO_REAL(MID(DataStr_Rear[3], 1, 16));	
	
	END_IF
	
	AccY_Rear	:=  AccY_Rear + (0.01 * STRING_TO_REAL(MID(DataStr_Rear[3], 2, 13))) +  (0.0001 * STRING_TO_REAL(MID(DataStr_Rear[3], 2, 11)));
	IF MID(DataStr_Rear[3], 1, 15) = '1' THEN
		AccY_Rear	:= AccY_Rear * (-1);
		
	END_IF
	
	(* parse accz *)
	IF MID(DataStr_Rear[3], 1, 10) = 'A' THEN
		AccZ_Rear	:= 10;
		
	ELSIF MID(DataStr_Rear[3], 1, 10) = 'B' THEN
		AccZ_Rear	:= 11;
		
	ELSIF MID(DataStr_Rear[3], 1, 10) = 'C' THEN
		AccZ_Rear	:= 12;
		
	ELSIF MID(DataStr_Rear[3], 1, 10) = 'D' THEN
		AccZ_Rear	:= 13;
		
	ELSIF MID(DataStr_Rear[3], 1, 10) = 'E' THEN
		AccZ_Rear	:= 14;
	
	ELSIF MID(DataStr_Rear[3], 1, 10) = 'F' THEN
		AccZ_Rear	:= 15;
		
	ELSE
		AccZ_Rear	:= STRING_TO_REAL(MID(DataStr_Rear[3], 1, 10));	
	
	END_IF
	
	AccZ_Rear	:=  AccZ_Rear + (0.01 * STRING_TO_REAL(MID(DataStr_Rear[3], 2, 7))) +  (0.0001 * STRING_TO_REAL(MID(DataStr_Rear[3], 2, 5)));
	IF MID(DataStr_Rear[3], 1, 9) = '1' THEN
		AccZ_Rear	:= AccZ_Rear * (-1);
		
	END_IF
	
	(* detect road section *)
	//algorithm for road section detection
	
	Counter_Rear			:= Counter_Rear + 1;	
	
END_IF

IF NOT (GVL.Lead_Trailer_State = 8 OR GVL.Lead_Trailer_State = 17416) THEN
	Pitch_Lead	:= 0;
	Roll_Lead	:= 0;
	AccX_Lead	:= 0; 
	AccY_Lead	:= 0;
	AccZ_Lead	:= 0;

END_IF

IF NOT (GVL.Rear_Trailer_State = 8) THEN
	Pitch_Rear	:= 0;
	Roll_Rear	:= 0;
	AccX_Rear	:= 0; 
	AccY_Rear	:= 0;
	AccZ_Rear	:= 0;

END_IF

(* count total received data per second *)
IF pSec <> Background_Time.cSec THEN 
		Total_Lead 	:= Counter_Lead;
		Counter_Lead := 0;
		
		Total_Rear 	:= Counter_Rear;
		Counter_Rear := 0;
		
		pSec	:= Background_Time.cSec;
END_IF

END_PROGRAM

// ---- POUs/Vacuum_Buffer_IMU.TcPOU
PROGRAM Vacuum_Buffer_IMU
VAR
	fbSqlDatabase	: FB_SQLDatabaseEvt(sNetID := '', tTimeout := T#1000S);
	fbSqlCommand	: FB_SQLCommandEvt(sNetID := '', tTimeout := T#1000S);
	fbSqlResult		: FB_SQLResultEvt(sNetID :='', tTimeout   := T#1000S); 
	nState			: INT;
	sCmd			: STRING(500000);
	Vacuumed		: BOOL;
END_VAR

CASE nState OF
				
		0:
			(* connect to buffer_imu *)		
			IF fbSqlDatabase.Connect(2) THEN
				IF fbSqlDatabase.bError THEN
					nState := 255; 
				ELSE
					IF fbSqlDatabase.bConnected THEN
						nState := nState+1;
					END_IF 
				END_IF
			END_IF
			
		1:
			IF fbSqlDatabase.CreateCmd(ADR(fbSqlCommand)) THEN
				IF fbSqlDatabase.bError THEN
					nState := 255; 
				ELSE
					nState := nState+1; 
				END_IF
			END_IF
		
		2:	
			IF NOT Vacuumed THEN
				(* build query *)	
				sCmd	:= 'VACUUM';
				
				IF fbSQLCommand.Execute(ADR(sCmd), SIZEOF(sCmd)) THEN
					IF fbSQLCommand.bError THEN
						nState := 255; 
					ELSE
						nState 		:= nState+1; 
					END_IF
				END_IF
				
			ELSE 
				nState := nState+1;
			END_IF
			
		3:
			IF fbSqlDatabase.Disconnect() THEN
				IF fbSqlDatabase.bError THEN
					nState := 255;
				ELSE
					nState 		:= nState+1;
					Vacuumed 	:= TRUE;
				END_IF
			END_IF
			
		255:
			nState := 0;
			
END_CASE

END_PROGRAM

// ---- POUs/Vacuum_Buffer_IMU_2.TcPOU
PROGRAM Vacuum_Buffer_IMU_2
VAR
	fbSqlDatabase	: FB_SQLDatabaseEvt(sNetID := '', tTimeout := T#1000S);
	fbSqlCommand	: FB_SQLCommandEvt(sNetID := '', tTimeout := T#1000S);
	fbSqlResult		: FB_SQLResultEvt(sNetID :='', tTimeout   := T#1000S); 
	nState			: INT;
	sCmd			: STRING(500000);
	Vacuumed		: BOOL;
END_VAR

CASE nState OF
				
		0:
			(* connect to buffer_imu *)		
			IF fbSqlDatabase.Connect(5) THEN
				IF fbSqlDatabase.bError THEN
					nState := 255; 
				ELSE
					IF fbSqlDatabase.bConnected THEN
						nState := nState+1;
					END_IF 
				END_IF
			END_IF
			
		1:
			IF fbSqlDatabase.CreateCmd(ADR(fbSqlCommand)) THEN
				IF fbSqlDatabase.bError THEN
					nState := 255; 
				ELSE
					nState := nState+1; 
				END_IF
			END_IF
		
		2:	
			IF NOT Vacuumed THEN
				(* build query *)	
				sCmd	:= 'VACUUM';
				
				IF fbSQLCommand.Execute(ADR(sCmd), SIZEOF(sCmd)) THEN
					IF fbSQLCommand.bError THEN
						nState := 255; 
					ELSE
						nState 		:= nState+1; 
					END_IF
				END_IF
				
			ELSE 
				nState := nState+1;
			END_IF
			
		3:
			IF fbSqlDatabase.Disconnect() THEN
				IF fbSqlDatabase.bError THEN
					nState := 255;
				ELSE
					nState 		:= nState+1;
					Vacuumed 	:= TRUE;
				END_IF
			END_IF
			
		255:
			nState := 0;
			
END_CASE

END_PROGRAM

// ---- POUs/Get_IMU.TcPOU
PROGRAM Get_IMU
VAR
	fbSqlDatabase	: FB_SQLDatabaseEvt(sNetID := '', tTimeout := T#1000S);
	fbSqlCommand	: FB_SQLCommandEvt(sNetID := '', tTimeout := T#1000S);
	fbSqlCommand2	: FB_SQLCommandEvt(sNetID := '', tTimeout := T#1000S);
	fbSqlResult		: FB_SQLResultEvt(sNetID:='', tTimeout   := T#1000S); 
    aReadStruct		: ARRAY[1..2500] OF ST_SelectStructIMU;
	nState			: INT;
	sCmd			: STRING(20000);
	sCmd2			: STRING(20000);
	val1			: INT;
	val2			: INT;
	exec			: BOOL;
	diff			: BOOL;
	rel				: BOOL;
	exec2			: BOOL;
	diff2			: BOOL;	
	rel2			: BOOL;
	exec3			: BOOL;
	diff3			: BOOL;	
	rel3			: BOOL;
	
	count			: ULINT;
	Data_Length		: ULINT;
	datetime		: STRING;
	Done			: BOOL;
	Deleted			: BOOL := TRUE;
	i 				: ULINT;
	
	TimeStr			: ARRAY[1..2500] OF STRING;	
	Trailer_ID_Lead	: ARRAY[1..2500] OF STRING;
	Trailer_ID_Rear	: ARRAY[1..2500] OF STRING;
	Pitch_Lead		: ARRAY[1..2500] OF STRING;
	Roll_Lead		: ARRAY[1..2500] OF STRING;
	AccX_Lead		: ARRAY[1..2500] OF STRING;
	AccY_Lead		: ARRAY[1..2500] OF STRING;
	AccZ_Lead		: ARRAY[1..2500] OF STRING;
	Pitch_Rear		: ARRAY[1..2500] OF STRING;
	Roll_Rear		: ARRAY[1..2500] OF STRING;
	AccX_Rear		: ARRAY[1..2500] OF STRING;
	AccY_Rear		: ARRAY[1..2500] OF STRING;
	AccZ_Rear		: ARRAY[1..2500] OF STRING;
	
	Dbid			: UDINT;
	Switch			: BOOL;
	Pragma_Done		: BOOL;
	bDisconnect		: BOOL;
	
END_VAR

(* get new data only if prev data sent to aws & saved to localdb *)
IF Main_SendIMU.Saved THEN
	Done	:= FALSE;
	Deleted	:= FALSE;
	IF fbSqlDatabase.bConnected THEN
		nState 	:= 1;
	ELSE
		nState 	:= 0;
	END_IF
END_IF

IF Switch THEN
	IF Buffer_IMU.Dbid = Dbid AND Buffer_IMU.fbSqlDatabase.bConnected THEN
		Switch := FALSE;
	END_IF
	
ELSIF Buffer_IMU.Initialized AND Buffer_IMU.fbSqlDatabase.bConnected THEN
	
	CASE nState OF
		
		0:
			//choose db opposite of buffer
			IF Buffer_IMU.Dbid = 2 THEN
				Dbid := 5;
			ELSE
				Dbid := 2;
			END_IF
			
			IF fbSqlDatabase.Connect(Dbid) THEN
				IF fbSqlDatabase.bError THEN
					nState := 255;
				ELSE
					nState := nState + 1;
				END_IF
			END_IF
			
		1:
			IF fbSqlDatabase.CreateCmd(ADR(fbSqlCommand)) THEN
				IF fbSqlDatabase.bError THEN
					nState := 255; 
				ELSE
					nState := nState+1; 
				END_IF
			END_IF
			
		2:	(* execute pragmas *)
			IF NOT Pragma_Done THEN
				sCmd	:= 'PRAGMA journal_mode = WAL; PRAGMA synchronous = NORMAL; PRAGMA temp_store = MEMORY; PRAGMA mmap_size = 30000000000; PRAGMA page_size = 32768; PRAGMA locking_mode = EXCLUSIVE;';
			
				IF fbSQLCommand.Execute(ADR(sCmd), SIZEOF(sCmd)) THEN
					IF fbSQLCommand.bError THEN
						nState := 255; 
					ELSE
						nState 		:= nState+1; 
						Pragma_Done := TRUE;
					END_IF
				END_IF
			
			ELSE
				nState 		:= nState+1;
			END_IF
		
		3:	
			IF Deleted THEN
				nState := nState+1;
			ELSE
				(* delete saved data from buffer *)
				sCmd2	:= 'DELETE FROM buffer_imu WHERE datetime IN (SELECT datetime FROM buffer_imu ORDER BY datetime ASC LIMIT ';
				sCmd2	:= CONCAT(sCmd2, ULINT_TO_STRING(Data_Length));
				sCmd2	:= CONCAT(sCmd2, ');');
				
				IF fbSQLCommand.Execute(ADR(sCmd2), SIZEOF(sCmd2)) THEN
					IF fbSQLCommand.bError THEN
						nState := 255; 
					ELSE
						nState := nState+1; 
						Deleted := TRUE;
					END_IF
				END_IF
			END_IF
			
		4:	
			(* count no of records in buffer *)
			sCmd2 := 'SELECT COUNT(*) FROM `buffer_imu`';
			
			IF fbSQLCommand.ExecuteDataReturn(ADR(sCmd2), SIZEOF(sCmd2), ADR(fbSqlResult)) THEN
				IF fbSQLCommand.bError THEN
					nState := 255; 
				ELSE
					nState := nState+1; 
				END_IF
			END_IF
			
		5:	
			IF fbSqlResult.Read(0, 1, ADR(count), SIZEOF(count), TRUE, TRUE) THEN
				IF fbSqlResult.bError THEN
					nState := 255; 
				ELSE
					nState := nState+1; 
				END_IF
			END_IF
			
		6:
			IF fbSqlResult.Release() THEN
				IF fbSqlResult.bError THEN
					nState := 255;
				ELSE
					nState := nState + 1;
				END_IF
				
			END_IF
			
		7:
			(* determine no of records to select *)
			IF count = 0 THEN
				Data_Length := 0;
				nState := 13;
			
			ELSIF count < 1000 THEN
				Data_Length := count;
				nState := nState+1;
			
			ELSE
				Data_Length := 1000;
				nState := nState+1;
			
			END_IF
			
		8:	
			(* get records from buffer *)
			sCmd2 := 'SELECT * FROM `buffer_imu` ORDER BY datetime ASC LIMIT ';
			sCmd2 := CONCAT(sCmd2, ULINT_TO_STRING(Data_Length));
			
			IF fbSQLCommand.ExecuteDataReturn(ADR(sCmd2), SIZEOF(sCmd2), ADR(fbSqlResult)) THEN
				IF fbSQLCommand.bError THEN
					nState := 255; 
				ELSE
					nState := nState+1; 
				END_IF
			END_IF
			
		9:
			IF fbSqlResult.Read(0, ULINT_TO_UDINT(Data_Length), ADR(aReadStruct), SIZEOF(aReadStruct), TRUE, TRUE) THEN
				IF fbSqlResult.bError THEN
					nState := 255; 
				ELSE
					nState := nState+1; 
				END_IF
			END_IF
			
		10:
			IF fbSqlResult.Release() THEN
				IF fbSqlResult.bError THEN
					nState := 255;
				ELSE
					nState := nState+1;
				END_IF
			END_IF
		
		11:
			(* parse query result *)
			FOR i:=1 TO Data_Length BY 1 DO
				TimeStr[i]			:= aReadStruct[i].datetime;
				
				Trailer_ID_Lead[i]			:= LINT_TO_STRING(aReadStruct[i].trailer_id_lead);
				Trailer_ID_Rear[i]			:= LINT_TO_STRING(aReadStruct[i].trailer_id_rear);
				//RoadSec[i]				:= UINT_TO_STRING(aReadStruct[i].RoadSec);
				Pitch_Lead[i]				:= REAL_TO_STRING(aReadStruct[i].pitch_lead);
				Roll_Lead[i]				:= REAL_TO_STRING(aReadStruct[i].roll_lead);
				AccX_Lead[i]				:= REAL_TO_STRING(aReadStruct[i].ax_lead);
				AccY_Lead[i]				:= REAL_TO_STRING(aReadStruct[i].ay_lead);
				AccZ_Lead[i]				:= REAL_TO_STRING(aReadStruct[i].az_lead);
				Pitch_Rear[i]				:= REAL_TO_STRING(aReadStruct[i].pitch_rear);
				Roll_Rear[i]				:= REAL_TO_STRING(aReadStruct[i].roll_rear);
				AccX_Rear[i]				:= REAL_TO_STRING(aReadStruct[i].ax_rear);
				AccY_Rear[i]				:= REAL_TO_STRING(aReadStruct[i].ay_rear);
				AccZ_Rear[i]				:= REAL_TO_STRING(aReadStruct[i].az_rear);
				
			END_FOR
			
			nState	:= nState + 1;
			
		12:
			Done	:= TRUE;
			
		13:	(* execute pragma optimize *)
			sCmd	:= 'PRAGMA optimize;';
			
			IF fbSQLCommand.Execute(ADR(sCmd), SIZEOF(sCmd)) THEN
				IF fbSQLCommand.bError THEN
					nState := 255; 
				ELSE
					nState := nState+1; 
				END_IF
			END_IF
			
		14:
			//disconnect from db
			IF bDisconnect := fbSqlDatabase.Disconnect() THEN
				IF fbSqlDatabase.bError THEN
					nState := 255;
				ELSE
					nState 		:= 0;
					Switch 		:= TRUE;
					Pragma_Done	:= FALSE;
				END_IF
			END_IF			
		
		255:
			nState	:= 0;	
			
	END_CASE
	
END_IF

END_PROGRAM

// ---- POUs/Main_SendIMU.TcPOU
PROGRAM Main_SendIMU
VAR
	Done		: BOOL;
	Sent		: BOOL;
	New_Data	: BOOL;
	Saved		: BOOL;
END_VAR

(* get data from database *)
Get_IMU();

IF New_Data := Get_IMU.Done THEN
	(* send data to aws iot core *)
	IF NOT Sent THEN
		Send_IMU();
		
		IF Send_IMU.Published THEN
			Sent	:= TRUE;
		END_IF	
		
	END_IF
	
	(* save data to localdb *)
	IF Sent THEN
		Save_IMU();
		
		IF Save_IMU.Done THEN
			Saved := TRUE;
		END_IF	
		
	END_IF
	
ELSE
	Sent	:= FALSE;
	Saved 	:= FALSE;
	
END_IF

END_PROGRAM

// ---- POUs/Send_IMU.TcPOU
PROGRAM Send_IMU
VAR
	fbMqttClient : FB_IotMqttClient;
	bSetParameter : BOOL := TRUE;
	bConnect : BOOL := TRUE;
	
	(* aws certificates *)
	
	(*-------------- actual ------------------*)
	(*
	rootCA		: STRING(255) := 'C:\Users\Administrator\Downloads\AWSCert\AmazonRootCA1.pem';
	thingCert	: STRING(255) := 'C:\Users\Administrator\Downloads\AWSCert\a2ca8bd1ed97a43e38f2bffcdf7ca64a29d3483826fdb03b3eb616af8a5efc9e-certificate.pem.crt';
	privateKey	: STRING(255) := 'C:\Users\Administrator\Downloads\AWSCert\a2ca8bd1ed97a43e38f2bffcdf7ca64a29d3483826fdb03b3eb616af8a5efc9e-private.pem.key';
	*)
	
	rootCA		: STRING(255) := 'C:\Users\Administrator\Downloads\AWSCert\AmazonRootCA1.pem';
	thingCert	: STRING(255) := 'C:\Users\Administrator\Downloads\AWSCert\8872c9f9d2c9335079f20c0506a3dd3599fd4d8552622bd2d7f8ae6d1681c64f-certificate.pem.crt';
	privateKey	: STRING(255) := 'C:\Users\Administrator\Downloads\AWSCert\8872c9f9d2c9335079f20c0506a3dd3599fd4d8552622bd2d7f8ae6d1681c64f-private.pem.key';
	
	(* ---------------- test ------------------- *)
	(*
	rootCA		: STRING(255) := 'C:\Users\muhammad.rahman\Downloads\double-sdt-test-certs\AmazonRootCA1.pem';
	thingCert	: STRING(255) := 'C:\Users\muhammad.rahman\Downloads\double-sdt-test-certs\8872c9f9d2c9335079f20c0506a3dd3599fd4d8552622bd2d7f8ae6d1681c64f-certificate.pem.crt';
	privateKey	: STRING(255) := 'C:\Users\muhammad.rahman\Downloads\double-sdt-test-certs\8872c9f9d2c9335079f20c0506a3dd3599fd4d8552622bd2d7f8ae6d1681c64f-private.pem.key';
	*)
	
	(* broker settings *)
	endpoint	: STRING := 'a2o01t3xth0mr1-ats.iot.ap-southeast-1.amazonaws.com';
	port		: UINT := 8883;
	//clientID	: STRING := 'double-sdt-1';
	clientID	: STRING := 'double-sdt-test';
	
	(* published message *)
	sTopicPub 		: STRING(255) := 'iot/smartproduct/mifa/double-sdt/imu'; //message topic
	sPayloadPub 	: STRING(50000000);
	str				: STRING(10000000);
	valSeparator	: STRING := '","';
	comma			: STRING := ',';
	arrayEnd		: STRING := '"]';
	arrayEnd2		: STRING := ']';
	msgEnd			: STRING := '}';
	i				: UDINT;
	
	(* topic subscription *)
	bSubscribed : BOOL;
	sTopicSub 	: STRING(255) := 'iot/smartproduct/mifa/double-sdt/imu';
	
	(* received message *)	
	{attribute 'TcEncoding':='UTF-8'}
	sTopicRcv : STRING(255);
	{attribute 'TcEncoding':='UTF-8'}
	sPayloadRcv : STRING(255);
	
	fbMessageQueue : FB_IotMqttMessageQueue;
	fbMessage : FB_IotMqttMessage;
	
	hrErrorOccurred : HRESULT; // contains the latest occurred error
	Published		: BOOL;
	Publish			: BOOL;
END_VAR

IF Main_SendIMU.New_Data THEN
	Publish		:= FALSE;
	Published 	:= FALSE;	
END_IF


IF bSetParameter THEN
	bSetParameter := FALSE;
	
	(* TLS settings for AWS IoT connection *)
	fbMqttClient.stTLS.sCA 		:= rootCA; //root CA
    fbMqttClient.stTLS.sCert 	:= thingCert; //certificate of thing
    fbMqttClient.stTLS.sKeyFile := privateKey; //private key of thing
	
	(* Broker settings für AWS IoT *)
	fbMqttClient.sHostName:= endpoint; //broker endpoint
	fbMqttClient.nHostPort:= port; //default mqtt tls port
	fbMqttClient.sClientId:= clientID; //client id
	fbMqttClient.sTopicPrefix:= ''; 
	
	fbMqttClient.ipMessageQueue := fbMessageQueue;
END_IF

(* connect to mqtt broker *)
fbMqttClient.Execute(bConnect); 
IF fbMqttClient.bError THEN
	// add your error logging here
	hrErrorOccurred := fbMqttClient.hrErrorCode;
END_IF

(* get message from subscribed topic *)
IF fbMessageQueue.nQueuedMessages > 0 THEN
	IF fbMessageQueue.Dequeue(fbMessage:=fbMessage) THEN
		fbMessage.GetTopic(pTopic:=ADR(sTopicRcv), nTopicSize:=SIZEOF(sTopicRcv) );
		fbMessage.GetPayload(pPayload:=ADR(sPayloadRcv), nPayloadSize:=SIZEOF(sPayloadRcv), bSetNullTermination:=FALSE);
	END_IF
END_IF

IF fbMqttClient.bConnected THEN	
	IF NOT bSubscribed THEN
		bSubscribed := fbMqttClient.Subscribe(sTopic:=sTopicSub, eQoS:=TcIotMqttQos.AtMostOnceDelivery); //subscribe to topic
		IF fbMqttClient.bError THEN
			// add your error logging here
			hrErrorOccurred := fbMqttClient.hrErrorCode;
		END_IF
	END_IF
	
	(* build message payload *)
	sPayloadPub := CONCAT('{"primemover_id":', Read_ID.PrimeMover_ID);
	
	(* lead trailer id string *)
	str	:= ',"trailer_id_lead":[';
	FOR i:=1 TO Get_IMU.Data_Length BY 1 DO
		CONCAT2(ADR(str), ADR(Get_IMU.Trailer_ID_Lead[i]), ADR(str), SIZEOF(str)); 
		
		IF i <> Get_IMU.Data_Length THEN
			CONCAT2(ADR(str), ADR(comma), ADR(str), SIZEOF(str));
		ELSE
			CONCAT2(ADR(str), ADR(arrayEnd2), ADR(str), SIZEOF(str));
		END_IF
		
	END_FOR
	
	CONCAT2(ADR(sPayloadPub), ADR(str), ADR(sPayloadPub), SIZEOF(sPayloadPub));
	
	(* rear trailer id string *)
	str	:= ',"trailer_id_rear":[';
	FOR i:=1 TO Get_IMU.Data_Length BY 1 DO
		CONCAT2(ADR(str), ADR(Get_IMU.Trailer_ID_Rear[i]), ADR(str), SIZEOF(str)); 
		
		IF i <> Get_IMU.Data_Length THEN
			CONCAT2(ADR(str), ADR(comma), ADR(str), SIZEOF(str));
		ELSE
			CONCAT2(ADR(str), ADR(arrayEnd2), ADR(str), SIZEOF(str));
		END_IF
		
	END_FOR
	
	CONCAT2(ADR(sPayloadPub), ADR(str), ADR(sPayloadPub), SIZEOF(sPayloadPub));
	
	(* date time string *)
	str	:= ',"datetime":["';
	FOR i:=1 TO Get_IMU.Data_Length BY 1 DO
		CONCAT2(ADR(str), ADR(Get_IMU.TimeStr[i]), ADR(str), SIZEOF(str)); 
		
		IF i <> Get_IMU.Data_Length THEN
			CONCAT2(ADR(str), ADR(valSeparator), ADR(str), SIZEOF(str));
		ELSE
			CONCAT2(ADR(str), ADR(arrayEnd), ADR(str), SIZEOF(str));
		END_IF
		
	END_FOR
	
	CONCAT2(ADR(sPayloadPub), ADR(str), ADR(sPayloadPub), SIZEOF(sPayloadPub));
	
	(* lead pitch string *)
	str	:= ',"pitch_lead":[';
	FOR i:=1 TO Get_IMU.Data_Length BY 1 DO
		CONCAT2(ADR(str), ADR(Get_IMU.Pitch_Lead[i]), ADR(str), SIZEOF(str)); 
		
		IF i <> Get_IMU.Data_Length THEN
			CONCAT2(ADR(str), ADR(comma), ADR(str), SIZEOF(str));
		ELSE
			CONCAT2(ADR(str), ADR(arrayEnd2), ADR(str), SIZEOF(str));
		END_IF
		
	END_FOR
	
	CONCAT2(ADR(sPayloadPub), ADR(str), ADR(sPayloadPub), SIZEOF(sPayloadPub));
	
	(* lead roll string *)
	str	:= ',"roll_lead":[';
	FOR i:=1 TO Get_IMU.Data_Length BY 1 DO
		CONCAT2(ADR(str), ADR(Get_IMU.Roll_Lead[i]), ADR(str), SIZEOF(str)); 
		
		IF i <> Get_IMU.Data_Length THEN
			CONCAT2(ADR(str), ADR(comma), ADR(str), SIZEOF(str));
		ELSE
			CONCAT2(ADR(str), ADR(arrayEnd2), ADR(str), SIZEOF(str));
		END_IF
		
	END_FOR
	
	CONCAT2(ADR(sPayloadPub), ADR(str), ADR(sPayloadPub), SIZEOF(sPayloadPub));
	
	(* lead acceleration x string *)
	str	:= ',"ax_lead":[';
	FOR i:=1 TO Get_IMU.Data_Length BY 1 DO
		CONCAT2(ADR(str), ADR(Get_IMU.AccX_Lead[i]), ADR(str), SIZEOF(str)); 
		
		IF i <> Get_IMU.Data_Length THEN
			CONCAT2(ADR(str), ADR(comma), ADR(str), SIZEOF(str));
		ELSE
			CONCAT2(ADR(str), ADR(arrayEnd2), ADR(str), SIZEOF(str));
		END_IF
		
	END_FOR
	
	CONCAT2(ADR(sPayloadPub), ADR(str), ADR(sPayloadPub), SIZEOF(sPayloadPub));
	
	(* lead acceleration y string *)
	str	:= ',"ay_lead":[';
	FOR i:=1 TO Get_IMU.Data_Length BY 1 DO
		CONCAT2(ADR(str), ADR(Get_IMU.AccY_Lead[i]), ADR(str), SIZEOF(str)); 
		
		IF i <> Get_IMU.Data_Length THEN
			CONCAT2(ADR(str), ADR(comma), ADR(str), SIZEOF(str));
		ELSE
			CONCAT2(ADR(str), ADR(arrayEnd2), ADR(str), SIZEOF(str));
		END_IF
		
	END_FOR
	
	CONCAT2(ADR(sPayloadPub), ADR(str), ADR(sPayloadPub), SIZEOF(sPayloadPub));
	
	(* lead acceleration z string *)
	str	:= ',"az_lead":[';
	FOR i:=1 TO Get_IMU.Data_Length BY 1 DO
		CONCAT2(ADR(str), ADR(Get_IMU.AccZ_Lead[i]), ADR(str), SIZEOF(str)); 
		
		IF i <> Get_IMU.Data_Length THEN
			CONCAT2(ADR(str), ADR(comma), ADR(str), SIZEOF(str));
		ELSE
			CONCAT2(ADR(str), ADR(arrayEnd2), ADR(str), SIZEOF(str));
		END_IF
		
	END_FOR
	
	CONCAT2(ADR(sPayloadPub), ADR(str), ADR(sPayloadPub), SIZEOF(sPayloadPub));
	
	(* lead pitch string *)
	str	:= ',"pitch_rear":[';
	FOR i:=1 TO Get_IMU.Data_Length BY 1 DO
		CONCAT2(ADR(str), ADR(Get_IMU.Pitch_Rear[i]), ADR(str), SIZEOF(str)); 
		
		IF i <> Get_IMU.Data_Length THEN
			CONCAT2(ADR(str), ADR(comma), ADR(str), SIZEOF(str));
		ELSE
			CONCAT2(ADR(str), ADR(arrayEnd2), ADR(str), SIZEOF(str));
		END_IF
		
	END_FOR
	
	CONCAT2(ADR(sPayloadPub), ADR(str), ADR(sPayloadPub), SIZEOF(sPayloadPub));
	
	(* rear roll string *)
	str	:= ',"roll_rear":[';
	FOR i:=1 TO Get_IMU.Data_Length BY 1 DO
		CONCAT2(ADR(str), ADR(Get_IMU.Roll_Rear[i]), ADR(str), SIZEOF(str)); 
		
		IF i <> Get_IMU.Data_Length THEN
			CONCAT2(ADR(str), ADR(comma), ADR(str), SIZEOF(str));
		ELSE
			CONCAT2(ADR(str), ADR(arrayEnd2), ADR(str), SIZEOF(str));
		END_IF
		
	END_FOR
	
	CONCAT2(ADR(sPayloadPub), ADR(str), ADR(sPayloadPub), SIZEOF(sPayloadPub));
	
	(* rear acceleration x string *)
	str	:= ',"ax_rear":[';
	FOR i:=1 TO Get_IMU.Data_Length BY 1 DO
		CONCAT2(ADR(str), ADR(Get_IMU.AccX_Rear[i]), ADR(str), SIZEOF(str)); 
		
		IF i <> Get_IMU.Data_Length THEN
			CONCAT2(ADR(str), ADR(comma), ADR(str), SIZEOF(str));
		ELSE
			CONCAT2(ADR(str), ADR(arrayEnd2), ADR(str), SIZEOF(str));
		END_IF
		
	END_FOR
	
	CONCAT2(ADR(sPayloadPub), ADR(str), ADR(sPayloadPub), SIZEOF(sPayloadPub));
	
	(* rear acceleration y string *)
	str	:= ',"ay_rear":[';
	FOR i:=1 TO Get_IMU.Data_Length BY 1 DO
		CONCAT2(ADR(str), ADR(Get_IMU.AccY_Rear[i]), ADR(str), SIZEOF(str)); 
		
		IF i <> Get_IMU.Data_Length THEN
			CONCAT2(ADR(str), ADR(comma), ADR(str), SIZEOF(str));
		ELSE
			CONCAT2(ADR(str), ADR(arrayEnd2), ADR(str), SIZEOF(str));
		END_IF
		
	END_FOR
	
	CONCAT2(ADR(sPayloadPub), ADR(str), ADR(sPayloadPub), SIZEOF(sPayloadPub));
	
	(* rear acceleration z string *)
	str	:= ',"az_rear":[';
	FOR i:=1 TO Get_IMU.Data_Length BY 1 DO
		CONCAT2(ADR(str), ADR(Get_IMU.AccZ_Rear[i]), ADR(str), SIZEOF(str)); 
		
		IF i <> Get_IMU.Data_Length THEN
			CONCAT2(ADR(str), ADR(comma), ADR(str), SIZEOF(str));
		ELSE
			CONCAT2(ADR(str), ADR(arrayEnd2), ADR(str), SIZEOF(str));
		END_IF
		
	END_FOR
	
	CONCAT2(ADR(sPayloadPub), ADR(str), ADR(sPayloadPub), SIZEOF(sPayloadPub));
	
	CONCAT2(ADR(sPayloadPub), ADR(msgEnd), ADR(sPayloadPub), SIZEOF(sPayloadPub)); //message ending
	
	(* publish message to subscribed topic *)
	IF Publish := fbMqttClient.Publish(sTopic:= sTopicPub, pPayload:= ADR(sPayloadPub), nPayloadSize:= LEN2(ADR(sPayloadPub)), eQoS:= TcIotMqttQos.AtMostOnceDelivery, bRetain:= FALSE, bQueue:= FALSE) THEN
		IF fbMqttClient.bError THEN
			// add your error logging here			
			hrErrorOccurred := fbMqttClient.hrErrorCode;
		ELSE
			Published 	:= TRUE;
		END_IF
		
	END_IF
	
END_IF

END_PROGRAM

// ---- POUs/Save_IMU.TcPOU
PROGRAM Save_IMU
VAR
	fbSqlDatabase	: FB_SQLDatabaseEvt(sNetID := '', tTimeout := T#1000S);
	fbSqlCommand	: FB_SQLCommandEvt(sNetID := '', tTimeout := T#1000S);
	fbSqlResult		: FB_SQLResultEvt(sNetID:='', tTimeout   := T#1000S); 
	sCmd			: STRING(1000000);
	sCmd2			: STRING(10000);
	nState			: INT := 9;
	
	Done			: BOOL;
	i				: ULINT;
	Vacuumed		: BOOL := FALSE;
	
	aReadStruct		: ST_SelectStructIMU;
	Oldest_data		: DWORD;
	Today			: DWORD;
	
	Deleted			: BOOL;
	Pragma_Done		: BOOL;
END_VAR

(* connect to localdb *)
IF NOT fbSqlDatabase.bConnected THEN
	
	IF Vacuum_IMU.Vacuumed THEN
		fbSqlDatabase.Connect(4);	
	END_IF
	
ELSE

	CASE nState OF
				
		0:
			Done := FALSE;
			IF fbSqlDatabase.CreateCmd(ADR(fbSqlCommand)) THEN
				IF fbSqlDatabase.bError THEN
					nState := 255; 
				ELSE
					IF NOT Deleted THEN
						nState := nState+1;
					ELSE
						nState := 6; //skip to save data
					END_IF
				END_IF
			END_IF
			
		1:	(* execute pragmas *)
			IF NOT Pragma_Done THEN
				sCmd	:= 'PRAGMA journal_mode = WAL; PRAGMA synchronous = NORMAL; PRAGMA temp_store = MEMORY; PRAGMA mmap_size = 30000000000; PRAGMA page_size = 32768; PRAGMA locking_mode = EXCLUSIVE;';
			
				IF fbSQLCommand.Execute(ADR(sCmd), SIZEOF(sCmd)) THEN
					IF fbSQLCommand.bError THEN
						nState := 255; 
					ELSE
						nState 		:= nState+1; 
						Pragma_Done := TRUE;
					END_IF
				END_IF
			
			ELSE
				nState 		:= nState+1;
			END_IF
			
		2:
			(* select oldest data from buffer_imu *)
			sCmd	:= 'SELECT * FROM `imu` ORDER BY datetime ASC LIMIT 1';
			
			IF fbSQLCommand.ExecuteDataReturn(ADR(sCmd), SIZEOF(sCmd), ADR(fbSqlResult)) THEN
				IF fbSQLCommand.bError THEN
					nState := 255; 
				ELSE
					nState := nState+1; 
				END_IF
			END_IF
			
		3:
			IF fbSqlResult.Read(0, 1, ADR(aReadStruct), SIZEOF(aReadStruct), TRUE, TRUE) THEN
				IF fbSqlResult.bError THEN
					nState := 255; 
				ELSE
					nState := nState+1; 
				END_IF
			END_IF
			
		4:
			IF fbSqlResult.Release() THEN
				IF fbSqlResult.bError THEN
					nState := 255;
				ELSE
					nState := nState+1;
				END_IF
			END_IF
			
		5:	
			//oldest data < today - 3 months?
			aReadStruct.datetime 	:= REPLACE(aReadStruct.datetime, '-', 1, 11);
			Oldest_data				:= DT_TO_DWORD(SYSTEMTIME_TO_DT(STRING_TO_SYSTEMTIME(aReadStruct.datetime)));
			Today					:= DT_TO_DWORD(SYSTEMTIME_TO_DT(Background_Time.fbTime.systemTime));
			
			IF Oldest_data < (Today - 7776000) THEN
				sCmd	:= 'DELETE FROM imu WHERE datetime < datetime($'now$', $'-3 month$');';
		
				IF fbSQLCommand.Execute(ADR(sCmd), SIZEOF(sCmd)) THEN
					IF fbSQLCommand.bError THEN
						nState := 255; 
					ELSE
						nState 	:= nState+1;
						Deleted	:= TRUE;
					END_IF
					
				END_IF
			ELSE
				nState 	:= nState+1;
				Deleted	:= TRUE;
			END_IF
			
		6:	
			(* build query *)	
			sCmd	:= 'INSERT INTO imu (datetime,trailer_id_lead,trailer_id_rear,pitch_lead,roll_lead,ax_lead,ay_lead,az_lead,pitch_rear,roll_rear,ax_rear,ay_rear,az_rear) VALUES ';
			
			FOR i := 1 TO Get_IMU.Data_Length BY 1 DO
					sCmd2:= CONCAT('($'', Get_IMU.TimeStr[i]);
					sCmd2:= CONCAT(sCmd2, '$',');
					sCmd2:= CONCAT(sCmd2, Get_IMU.Trailer_ID_Lead[i]);
					sCmd2:= CONCAT(sCmd2, ',');
					sCmd2:= CONCAT(sCmd2, Get_IMU.Trailer_ID_Rear[i]);
					sCmd2:= CONCAT(sCmd2, ',');
					sCmd2:= CONCAT(sCmd2, Get_IMU.Pitch_Lead[i]);
					sCmd2:= CONCAT(sCmd2, ',');
					sCmd2:= CONCAT(sCmd2, Get_IMU.Roll_Lead[i]);
					sCmd2:= CONCAT(sCmd2, ',');
					sCmd2:= CONCAT(sCmd2, Get_IMU.AccX_Lead[i]);
					sCmd2:= CONCAT(sCmd2, ',');
					sCmd2:= CONCAT(sCmd2, Get_IMU.AccY_Lead[i]);
					sCmd2:= CONCAT(sCmd2, ',');
					sCmd2:= CONCAT(sCmd2, Get_IMU.AccZ_Lead[i]);
					sCmd2:= CONCAT(sCmd2, ',');
					sCmd2:= CONCAT(sCmd2, Get_IMU.Pitch_Rear[i]);
					sCmd2:= CONCAT(sCmd2, ',');
					sCmd2:= CONCAT(sCmd2, Get_IMU.Roll_Rear[i]);
					sCmd2:= CONCAT(sCmd2, ',');
					sCmd2:= CONCAT(sCmd2, Get_IMU.AccX_Rear[i]);
					sCmd2:= CONCAT(sCmd2, ',');
					sCmd2:= CONCAT(sCmd2, Get_IMU.AccY_Rear[i]);
					sCmd2:= CONCAT(sCmd2, ',');
					sCmd2:= CONCAT(sCmd2, Get_IMU.AccZ_Rear[i]);
					
					IF i = Get_IMU.Data_Length THEN
						sCmd2:= CONCAT(sCmd2, ')');
					ELSE	
						sCmd2:= CONCAT(sCmd2, '),');
					END_IF
					
					CONCAT2(ADR(sCmd), ADR(sCmd2), ADR(sCmd), SIZEOF(sCmd));
				END_FOR
			
			IF fbSQLCommand.Execute(ADR(sCmd), SIZEOF(sCmd)) THEN
				IF fbSQLCommand.bError THEN
					nState := 255; 
				ELSE
					nState := nState+1; 
				END_IF
				
			END_IF
		
		7: 
			Done	:= TRUE;
			nState	:= nState + 1;
			
		8:
			IF NOT Main_Send.New_IMU THEN
				nState := nState + 1;
			END_IF
			
		9:
			IF Main_Send.Sent THEN
				nState := 0;
			END_IF
				
		255:
			nState := 0;
	
	END_CASE
	
END_IF

END_PROGRAM

// ---- POUs/Vacuum_IMU.TcPOU
PROGRAM Vacuum_IMU
VAR
	fbSqlDatabase	: FB_SQLDatabaseEvt(sNetID := '', tTimeout := T#1000S);
	fbSqlCommand	: FB_SQLCommandEvt(sNetID := '', tTimeout := T#1000S);
	fbSqlResult		: FB_SQLResultEvt(sNetID :='', tTimeout   := T#1000S); 
	nState			: INT;
	sCmd			: STRING(500000);
	Vacuumed		: BOOL;
END_VAR

CASE nState OF
				
		0:
			(* connect to buffer_imu *)		
			IF fbSqlDatabase.Connect(4) THEN
				IF fbSqlDatabase.bError THEN
					nState := 255; 
				ELSE
					IF fbSqlDatabase.bConnected THEN
						nState := nState+1;
					END_IF 
				END_IF
			END_IF
			
		1:
			IF fbSqlDatabase.CreateCmd(ADR(fbSqlCommand)) THEN
				IF fbSqlDatabase.bError THEN
					nState := 255; 
				ELSE
					nState := nState+1; 
				END_IF
			END_IF
			
		2:	(* execute pragmas *)
			sCmd	:= 'PRAGMA journal_mode = WAL; PRAGMA synchronous = NORMAL; PRAGMA temp_store = MEMORY; PRAGMA mmap_size = 30000000000; PRAGMA page_size = 32768; PRAGMA locking_mode = EXCLUSIVE;';
			
			IF fbSQLCommand.Execute(ADR(sCmd), SIZEOF(sCmd)) THEN
				IF fbSQLCommand.bError THEN
					nState := 255; 
				ELSE
					nState := nState+1; 
				END_IF
			END_IF
		
		3:	
			IF NOT Vacuumed THEN
				(* build query *)	
				sCmd	:= 'VACUUM';
				
				IF fbSQLCommand.Execute(ADR(sCmd), SIZEOF(sCmd)) THEN
					IF fbSQLCommand.bError THEN
						nState := 255; 
					ELSE
						nState 		:= nState+1; 
					END_IF
				END_IF
				
			ELSE 
				nState := nState+1;
			END_IF
			
		4:	(* execute pragma optimize *)
			sCmd	:= 'PRAGMA optimize;';
			
			IF fbSQLCommand.Execute(ADR(sCmd), SIZEOF(sCmd)) THEN
				IF fbSQLCommand.bError THEN
					nState := 255; 
				ELSE
					nState := nState+1; 
				END_IF
			END_IF
		
		5:
			IF fbSqlDatabase.Disconnect() THEN
				IF fbSqlDatabase.bError THEN
					nState := 255;
				ELSE
					nState 		:= nState+1;
					Vacuumed 	:= TRUE;
				END_IF
			END_IF
			
		255:
			nState := 0;
			
END_CASE

END_PROGRAM

// ---- POUs/Main_Send.TcPOU
PROGRAM Main_Send
VAR
END_VAR

Main_SendData();
Main_SendIMU();
;

END_PROGRAM

// ---- POUs/Main_SendData.TcPOU
PROGRAM Main_SendData
VAR	
	Done		: BOOL;
	Sent		: BOOL;
	New_Data	: BOOL;
	Saved		: BOOL;
END_VAR

(* get data from database *)
Get_Data();
 
IF New_Data := Get_Data.Done THEN
	(* send data to aws iot core *)
	IF NOT Sent THEN
		Send_Data();
		
		IF Send_Data.Published THEN
			Sent	:= TRUE;
		END_IF	
		
	END_IF
	
	(* save data to localdb *)
	IF Sent THEN
		Save_Data();
		
		IF Save_Data.Done THEN
			Saved := TRUE;
		END_IF	
		
	END_IF
	
ELSE
	Sent	:= FALSE;
	Saved 	:= FALSE;
	
END_IF

END_PROGRAM

// ---- POUs/Get_Data.TcPOU
PROGRAM Get_Data
VAR
	fbSqlDatabase	: FB_SQLDatabaseEvt(sNetID := '', tTimeout := T#1000S);
	fbSqlCommand	: FB_SQLCommandEvt(sNetID := '', tTimeout := T#1000S);
	fbSqlCommand2	: FB_SQLCommandEvt(sNetID := '', tTimeout := T#1000S);
	fbSqlResult		: FB_SQLResultEvt(sNetID:='', tTimeout   := T#1000S); 
    aReadStruct		: ARRAY[1..50] OF ST_SelectStructData;
	nState			: INT;
	sCmd			: STRING(20000);
	sCmd2			: STRING(20000);
	
	count			: ULINT;
	Data_Length		: ULINT;
	datetime		: STRING;
	Done			: BOOL;
	Deleted			: BOOL := TRUE;
	i 				: ULINT;
	
	TimeStr				: ARRAY[1..50] OF STRING;	
	Trailer_ID_Lead		: ARRAY[1..50] OF STRING;
	Trailer_ID_Rear		: ARRAY[1..50] OF STRING;
	Lat					: ARRAY[1..50] OF STRING;
	Lon					: ARRAY[1..50] OF STRING;
	Speed				: ARRAY[1..50] OF STRING;
	Overspeed			: ARRAY[1..50] OF STRING;
	Payload_Lead		: ARRAY[1..50] OF STRING;
	Payload_Rear		: ARRAY[1..50] OF STRING;
	Overload_Lead		: ARRAY[1..50] OF STRING;
	Overload_Rear		: ARRAY[1..50] OF STRING;
	Pressure_Lead		: ARRAY[1..50] OF STRING;
	Pressure_Rear		: ARRAY[1..50] OF STRING;
	Overpressure_Lead	: ARRAY[1..50] OF STRING;
	Overpressure_Rear	: ARRAY[1..50] OF STRING;
	EventCode			: ARRAY[1..50] OF STRING;
	
	Dbid			: UDINT;
	Switch			: BOOL;
	Pragma_Done		: BOOL;
	bDisconnect		: BOOL;
END_VAR

(* get new data only if prev data sent to aws & saved to localdb *)
IF Main_SendData.Saved THEN
	Done	:= FALSE;
	Deleted	:= FALSE;
	IF fbSqlDatabase.bConnected THEN
		nState 	:= 1;
	ELSE
		nState 	:= 0;
	END_IF
END_IF

IF Switch THEN
	IF Buffer_Data.Dbid = Dbid AND Buffer_Data.fbSqlDatabase.bConnected THEN
		Switch := FALSE;
	END_IF
	
ELSIF Buffer_Data.Initialized AND Buffer_Data.fbSqlDatabase.bConnected THEN
	
	CASE nState OF
		
		0:
			//choose db opposite of buffer
			IF Buffer_Data.Dbid = 1 THEN
				Dbid := 6;
			ELSE
				Dbid := 1;
			END_IF
			
			IF fbSqlDatabase.Connect(Dbid) THEN
				IF fbSqlDatabase.bError THEN
					nState := 255;
				ELSE
					nState := nState + 1;
				END_IF
			END_IF
			
		1:
			IF fbSqlDatabase.CreateCmd(ADR(fbSqlCommand)) THEN
				IF fbSqlDatabase.bError THEN
					nState := 255; 
				ELSE
					nState := nState+1; 
				END_IF
			END_IF
			
		2:	(* execute pragmas *)
			IF NOT Pragma_Done THEN
				sCmd	:= 'PRAGMA journal_mode = WAL; PRAGMA synchronous = NORMAL; PRAGMA temp_store = MEMORY; PRAGMA mmap_size = 30000000000; PRAGMA page_size = 32768; PRAGMA locking_mode = EXCLUSIVE;';
			
				IF fbSQLCommand.Execute(ADR(sCmd), SIZEOF(sCmd)) THEN
					IF fbSQLCommand.bError THEN
						nState := 255; 
					ELSE
						nState 		:= nState+1; 
						Pragma_Done := TRUE;
					END_IF
				END_IF
			
			ELSE
				nState 		:= nState+1;
			END_IF
		
		3:	
			IF Deleted THEN
				nState := nState+1;
			ELSE
				(* delete saved data from buffer *)
				sCmd2	:= 'DELETE FROM buffer_data WHERE datetime IN (SELECT datetime FROM buffer_data ORDER BY datetime ASC LIMIT ';
				sCmd2	:= CONCAT(sCmd2, ULINT_TO_STRING(Data_Length));
				sCmd2	:= CONCAT(sCmd2, ');');
				
				IF fbSQLCommand.Execute(ADR(sCmd2), SIZEOF(sCmd2)) THEN
					IF fbSQLCommand.bError THEN
						nState := 255; 
					ELSE
						nState := nState+1; 
						Deleted := TRUE;
					END_IF
				END_IF
			END_IF
			
		4:	
			(* count no of records in buffer *)
			sCmd2 := 'SELECT COUNT(*) FROM `buffer_data`';
			
			IF fbSQLCommand.ExecuteDataReturn(ADR(sCmd2), SIZEOF(sCmd2), ADR(fbSqlResult)) THEN
				IF fbSQLCommand.bError THEN
					nState := 255; 
				ELSE
					nState := nState+1; 
				END_IF
			END_IF
			
		5:	
			IF fbSqlResult.Read(0, 1, ADR(count), SIZEOF(count), TRUE, TRUE) THEN
				IF fbSqlResult.bError THEN
					nState := 255; 
				ELSE
					nState := nState+1; 
				END_IF
			END_IF
			
		6:
			IF fbSqlResult.Release() THEN
				IF fbSqlResult.bError THEN
					nState := 255;
				ELSE
					nState := nState + 1;
				END_IF
				
			END_IF
			
		7:
			(* determine no of records to select *)
			IF count = 0 THEN
				Data_Length := 0;
				nState := 13;
			
			ELSIF count < 50 THEN
				Data_Length := count;
				nState := nState+1;
			
			ELSE
				Data_Length := 50;
				nState := nState+1;
			
			END_IF
			
		8:	
			(* get records from buffer *)
			sCmd2 := 'SELECT * FROM `buffer_data` ORDER BY datetime ASC LIMIT ';
			sCmd2 := CONCAT(sCmd2, ULINT_TO_STRING(Data_Length));
			
			IF fbSQLCommand.ExecuteDataReturn(ADR(sCmd2), SIZEOF(sCmd2), ADR(fbSqlResult)) THEN
				IF fbSQLCommand.bError THEN
					nState := 255; 
				ELSE
					nState := nState+1; 
				END_IF
			END_IF
			
		9:
			IF fbSqlResult.Read(0, ULINT_TO_UDINT(Data_Length), ADR(aReadStruct), SIZEOF(aReadStruct), TRUE, TRUE) THEN
				IF fbSqlResult.bError THEN
					nState := 255; 
				ELSE
					nState := nState+1; 
				END_IF
			END_IF
			
		10:
			IF fbSqlResult.Release() THEN
				IF fbSqlResult.bError THEN
					nState := 255;
				ELSE
					nState := nState+1;
				END_IF
			END_IF
		
		11:
			(* parse query result *)
			FOR i:=1 TO Data_Length BY 1 DO
				TimeStr[i] 					:= aReadStruct[i].datetime;
				Trailer_ID_Lead[i] 			:= LINT_TO_STRING(aReadStruct[i].trailer_id_lead);
				Trailer_ID_Rear[i] 			:= LINT_TO_STRING(aReadStruct[i].trailer_id_rear);
				Lat[i] 						:= REAL_TO_STRING(aReadStruct[i].latitude);
				Lon[i] 						:= REAL_TO_STRING(aReadStruct[i].longitude);
				Speed[i] 					:= REAL_TO_STRING(aReadStruct[i].speed);
				Overspeed[i] 				:= LINT_TO_STRING(aReadStruct[i].overspeed);
				Payload_Lead[i]				:= REAL_TO_STRING(aReadStruct[i].payload_lead);
				Payload_Rear[i] 			:= REAL_TO_STRING(aReadStruct[i].payload_rear);
				Overload_Lead[i] 			:= LINT_TO_STRING(aReadStruct[i].overload_lead);
				Overload_Rear[i] 			:= LINT_TO_STRING(aReadStruct[i].overload_rear);
				Pressure_Lead[i] 			:= REAL_TO_STRING(aReadStruct[i].pressure_lead);
				Pressure_Rear[i] 			:= REAL_TO_STRING(aReadStruct[i].pressure_rear);
				Overpressure_Lead[i] 		:= REAL_TO_STRING(aReadStruct[i].overpressure_lead);
				Overpressure_Rear[i] 		:= REAL_TO_STRING(aReadStruct[i].overpressure_rear);
				EventCode[i]	 			:= REAL_TO_STRING(aReadStruct[i].event_code);
				
			END_FOR
			
			nState	:= nState + 1;
			
		12:
			Done	:= TRUE;
			
		13:	(* execute pragma optimize *)
			sCmd	:= 'PRAGMA optimize;';
			
			IF fbSQLCommand.Execute(ADR(sCmd), SIZEOF(sCmd)) THEN
				IF fbSQLCommand.bError THEN
					nState := 255; 
				ELSE
					nState := nState+1; 
				END_IF
			END_IF
			
		14:
			//disconnect from db
			IF bDisconnect := fbSqlDatabase.Disconnect() THEN
				IF fbSqlDatabase.bError THEN
					nState := 255;
				ELSE
					nState 		:= 0;
					Switch 		:= TRUE;
					Pragma_Done	:= FALSE;
				END_IF
			END_IF			
		
		255:
			nState	:= 0;	
			
	END_CASE
	
END_IF

END_PROGRAM

// ---- POUs/Buffer_Data.TcPOU
PROGRAM Buffer_Data
VAR
	pSec		: WORD;
	diff		: BOOL;
	
	TimeStr				: STRING;
	Trailer_ID_Lead		: STRING;
	Trailer_ID_Rear		: STRING;
	Lat					: STRING;
	Lon					: STRING;
	Speed				: STRING;
	Overspeed			: STRING;
	Payload_Lead		: STRING;
	Payload_Rear		: STRING;
	Overload_Lead		: STRING;
	Overload_Rear		: STRING;
	Pressure_Lead		: STRING;
	Pressure_Rear		: STRING;
	Overpressure_Lead	: STRING;
	Overpressure_Rear	: STRING;
	EventCode			: STRING;
	
	fbSqlDatabase	: FB_SQLDatabaseEvt(sNetID := '', tTimeout := T#1000S);
	fbSqlCommand	: FB_SQLCommandEvt(sNetID := '', tTimeout := T#1000S);
	fbSqlResult		: FB_SQLResultEvt(sNetID:='', tTimeout   := T#1000S); 
	sCmd			: STRING(10000);
	sCmd2			: STRING(10000);
	nState			: INT;
	nState_Switch	: INT;
	
	Buffer_Done		: BOOL;
	Done			: BOOL;
	Vacuumed		: BOOL := FALSE;
	
	Initialized 	: BOOL := FALSE;
	i				: INT;
	Pragma_Done		: BOOL;
	Counter			: ULINT;
	Dbid			: UDINT;
	bDisconnect		: BOOL;
	
	aReadStruct		: ST_SelectStructData;
	aReadStruct_2	: ST_SelectStructData;
	Timestamp		: DT;
	Timestamp_2		: DT; 
	
END_VAR

(* convert to strings *)
IF GVL.Lead_Trailer_State = 8 OR GVL.Lead_Trailer_State = 17416 THEN
	Trailer_ID_Lead		:= UINT_TO_STRING(Read_ID.Trailer_ID_Lead);
	Payload_Lead		:= REAL_TO_STRING(Read_Payload.Payload_Lead);
	Overload_Lead		:= BOOL_TO_STRING(Read_Payload.Overload_Lead);
	Pressure_Lead		:= REAL_TO_STRING(Read_Pressure.Pressure_Lead);
	Overpressure_Lead	:= BOOL_TO_STRING(Read_Pressure.Overpressure_Lead);
ELSE
	Trailer_ID_Lead		:= '99';
	Payload_Lead		:= '0';
	Overload_Lead		:= 'FALSE';
	Pressure_Lead		:= '0';
	Overpressure_Lead	:= 'FALSE';	
END_IF

IF GVL.Rear_Trailer_State = 8 THEN
	Trailer_ID_Rear		:= UINT_TO_STRING(Read_ID.Trailer_ID_Rear);
	Payload_Rear		:= REAL_TO_STRING(Read_Payload.Payload_Rear);
	Overload_Rear		:= BOOL_TO_STRING(Read_Payload.Overload_Rear);
	Pressure_Rear		:= REAL_TO_STRING(Read_Pressure.Pressure_Rear);
	Overpressure_Rear	:= BOOL_TO_STRING(Read_Pressure.Overpressure_Rear);
ELSE
	Trailer_ID_Rear		:= '99';
	Payload_Rear		:= '0';
	Overload_Rear		:= 'FALSE';
	Pressure_Rear		:= '0';
	Overpressure_Rear	:= 'FALSE';
END_IF

TimeStr				:= Main_Read.TimeStr;
TimeStr				:= REPLACE(TimeStr, ' ', 1, 11);
Lat					:= REAL_TO_STRING(Read_GPS.Lat);
Lon					:= REAL_TO_STRING(Read_GPS.Lon);
Speed				:= REAL_TO_STRING(Read_GPS.Speed);
Overspeed			:= BOOL_TO_STRING(Read_GPS.Overspeed);

IF Read_FatigueCam.New_Event THEN
	Buffer_Done := FALSE;
END_IF

EventCode	:= Read_FatigueCam.EventCode;

IF NOT Initialized THEN
	
	//initialization (choose which database for buffer)
	CASE nState OF
		
		0:
			(* connect to buffer_data *)	
			IF Vacuum_Buffer_Data.Vacuumed THEN
				
				Dbid := 1;		
				IF fbSqlDatabase.Connect(Dbid) THEN
					IF fbSqlDatabase.bError THEN
						nState := 255; 
					ELSE
						nState := nState+1;
					END_IF
				END_IF
				
			END_IF
			
			
		1:
			IF fbSqlDatabase.CreateCmd(ADR(fbSqlCommand)) THEN
				IF fbSqlDatabase.bError THEN
					nState := 255; 
				ELSE
					nState := nState+1; 
				END_IF
			END_IF
			
		2:	(* execute pragmas *)
			sCmd	:= 'PRAGMA journal_mode = WAL; PRAGMA synchronous = NORMAL; PRAGMA temp_store = MEMORY; PRAGMA mmap_size = 30000000000; PRAGMA page_size = 32768; PRAGMA locking_mode = EXCLUSIVE;';
			
			IF fbSQLCommand.Execute(ADR(sCmd), SIZEOF(sCmd)) THEN
				IF fbSQLCommand.bError THEN
					nState := 255; 
				ELSE
					nState := nState+1; 
				END_IF
			END_IF
			
		3:
			(* select oldest data from buffer_data *)
			sCmd	:= 'SELECT * FROM `buffer_data` ORDER BY datetime ASC LIMIT 1';
			
			IF fbSQLCommand.ExecuteDataReturn(ADR(sCmd), SIZEOF(sCmd), ADR(fbSqlResult)) THEN
				IF fbSQLCommand.bError THEN
					nState := 255; 
				ELSE
					nState := nState+1; 
				END_IF
			END_IF
			
		4:
			IF fbSqlResult.Read(0, 1, ADR(aReadStruct), SIZEOF(aReadStruct), TRUE, TRUE) THEN
				IF fbSqlResult.bError THEN
					nState := 255; 
				ELSE
					nState := nState+1; 
				END_IF
			END_IF
			
		5:
			IF fbSqlResult.Release() THEN
				IF fbSqlResult.bError THEN
					nState := 255;
				ELSE
					nState := nState+1;
				END_IF
			END_IF
			
		6:	(* execute pragma optimize *)
			sCmd	:= 'PRAGMA optimize;';
			
			IF fbSQLCommand.Execute(ADR(sCmd), SIZEOF(sCmd)) THEN
				IF fbSQLCommand.bError THEN
					nState := 255; 
				ELSE
					nState := nState+1; 
				END_IF
			END_IF
			
		7:
			(* disconnect from buffer_data *)
			IF fbSqlDatabase.Disconnect() THEN
				IF fbSqlDatabase.bError THEN
					nState := 255;
				ELSE
					nState := nState+1;
				END_IF
			END_IF
			
		8:	
			(* connect to buffer_data_2 *)
			IF Vacuum_Buffer_Data_2.Vacuumed THEN
				
				Dbid := 6;	
				IF fbSqlDatabase.Connect(Dbid) THEN
					IF fbSqlDatabase.bError THEN
						nState := 255; 
					ELSE
						nState := nState+1;
					END_IF
				END_IF
				
			END_IF	
			
		9:
			IF fbSqlDatabase.CreateCmd(ADR(fbSqlCommand)) THEN
				IF fbSqlDatabase.bError THEN
					nState := 255; 
				ELSE
					nState := nState+1; 
				END_IF
			END_IF
			
		10:	(* execute pragmas *)
			sCmd	:= 'PRAGMA journal_mode = WAL; PRAGMA synchronous = NORMAL; PRAGMA temp_store = MEMORY; PRAGMA mmap_size = 30000000000; PRAGMA page_size = 32768; PRAGMA locking_mode = EXCLUSIVE;';
			
			IF fbSQLCommand.Execute(ADR(sCmd), SIZEOF(sCmd)) THEN
				IF fbSQLCommand.bError THEN
					nState := 255; 
				ELSE
					nState := nState+1; 
				END_IF
			END_IF
			
		11:
			(* select oldest data from buffer_data *)
			sCmd	:= 'SELECT * FROM `buffer_data` ORDER BY datetime ASC LIMIT 1';
			
			IF fbSQLCommand.ExecuteDataReturn(ADR(sCmd), SIZEOF(sCmd), ADR(fbSqlResult)) THEN
				IF fbSQLCommand.bError THEN
					nState := 255; 
				ELSE
					nState := nState+1; 
				END_IF
			END_IF
			
		12:
			IF fbSqlResult.Read(0, 1, ADR(aReadStruct_2), SIZEOF(aReadStruct_2), TRUE, TRUE) THEN
				IF fbSqlResult.bError THEN
					nState := 255; 
				ELSE
					nState := nState+1; 
				END_IF
			END_IF
			
		13:
			IF fbSqlResult.Release() THEN
				IF fbSqlResult.bError THEN
					nState := 255;
				ELSE
					nState := nState+1;
				END_IF
			END_IF
			
		14:	(* execute pragma optimize *)
			sCmd	:= 'PRAGMA optimize;';
			
			IF fbSQLCommand.Execute(ADR(sCmd), SIZEOF(sCmd)) THEN
				IF fbSQLCommand.bError THEN
					nState := 255; 
				ELSE
					nState := nState+1; 
				END_IF
			END_IF
			
		15:
			(* disconnect from buffer_data_2 *)
			IF bDisconnect := fbSqlDatabase.Disconnect() THEN
				IF fbSqlDatabase.bError THEN
					nState := 255;
				ELSE
					nState := nState+1;
				END_IF
			END_IF
			
		16:
			// compare oldest data datetime
			aReadStruct.datetime 	:= REPLACE(aReadStruct.datetime, '-', 1, 11);
			aReadStruct_2.datetime 	:= REPLACE(aReadStruct_2.datetime, '-', 1, 11);
			
			Timestamp	:= SYSTEMTIME_TO_DT(STRING_TO_SYSTEMTIME(aReadStruct.datetime));
			Timestamp_2	:= SYSTEMTIME_TO_DT(STRING_TO_SYSTEMTIME(aReadStruct_2.datetime));

			IF Timestamp = DT#1970-1-1-00:00:00 THEN
				Dbid := 1;
			ELSIF Timestamp_2 = DT#1970-1-1-00:00:00 THEN
				Dbid := 6;
			ELSIF Timestamp > Timestamp_2 THEN
				Dbid := 1;
			ELSE
				Dbid := 6;
			END_IF
			
			Initialized := TRUE;
			nState		:= 0;
			
		255:
			nState := 0;
		
	END_CASE
	
ELSE
	
	(* save data to buffer every second *)
	IF diff:= Background_Time.cSec <> pSec THEN
		
		//database switching
		IF Get_Data.Switch AND Counter >= 5 THEN
			
			CASE nState_Switch OF
				
				0:	(* execute pragma optimize *)
					sCmd	:= 'PRAGMA optimize;';
					
					IF fbSQLCommand.Execute(ADR(sCmd), SIZEOF(sCmd)) THEN
						IF fbSQLCommand.bError THEN
							nState_Switch := 255; 
						ELSE
							nState_Switch := nState_Switch+1; 
						END_IF
					END_IF
				
				1:
					IF fbSqlDatabase.bConnected THEN
						fbSqlDatabase.Disconnect();
					ELSE
						IF Dbid = 1 THEN
							Dbid := 6;
						ELSE
							Dbid := 1;
						END_IF
						Counter			:= 0;
						nState_Switch 	:= 0;
						Pragma_Done		:= FALSE;
					END_IF
					
				255:
					nState_Switch := 0;
					
			END_CASE
		
		ELSE
			
			IF Done THEN
				Done	:= FALSE;
				IF fbSqlDatabase.bConnected THEN
					nState 	:= 1;
				ELSE
					nState 	:= 0;
				END_IF	
			END_IF
			
			CASE nState OF	
				0:	
					IF fbSqlDatabase.Connect(Dbid) THEN
						IF fbSqlDatabase.bError THEN
							nState := 255;
						ELSE
							nState := nState + 1; 
						END_IF
					END_IF
				
				1:
					IF fbSqlDatabase.CreateCmd(ADR(fbSqlCommand)) THEN
						IF fbSqlDatabase.bError THEN
							nState := 255; 
						ELSE
							nState := nState+1; 
						END_IF
					END_IF
					
				2:	(* execute pragmas *)
					IF NOT Pragma_Done THEN
						sCmd	:= 'PRAGMA journal_mode = WAL; PRAGMA synchronous = NORMAL; PRAGMA temp_store = MEMORY; PRAGMA mmap_size = 30000000000; PRAGMA page_size = 32768; PRAGMA locking_mode = EXCLUSIVE;';
					
						IF fbSQLCommand.Execute(ADR(sCmd), SIZEOF(sCmd)) THEN
							IF fbSQLCommand.bError THEN
								nState := 255; 
							ELSE
								nState 		:= nState+1; 
								Pragma_Done := TRUE;
							END_IF
						END_IF
					
					ELSE
						nState 		:= nState+1;
 
					END_IF
					
				3:	
					(* build query *)	
					sCmd:= 'INSERT INTO buffer_data (datetime,trailer_id_lead,trailer_id_rear,latitude,longitude,speed,overspeed,payload_lead,payload_rear,overload_lead,overload_rear,pressure_lead,pressure_rear,overpressure_lead,overpressure_rear,event_code) VALUES ($'';
					sCmd2:= TimeStr;
					sCmd2:= CONCAT(sCmd2, '$',');
					sCmd2:= CONCAT(sCmd2, Trailer_ID_Lead);
					sCmd2:= CONCAT(sCmd2, ',');
					sCmd2:= CONCAT(sCmd2, Trailer_ID_Rear);
					sCmd2:= CONCAT(sCmd2, ',');
					sCmd2:= CONCAT(sCmd2, Lat);
					sCmd2:= CONCAT(sCmd2, ',');
					sCmd2:= CONCAT(sCmd2, Lon);
					sCmd2:= CONCAT(sCmd2, ',');
					sCmd2:= CONCAT(sCmd2, Speed);
					sCmd2:= CONCAT(sCmd2, ',');
					sCmd2:= CONCAT(sCmd2, Overspeed);
					sCmd2:= CONCAT(sCmd2, ',');
					sCmd2:= CONCAT(sCmd2, Payload_Lead);
					sCmd2:= CONCAT(sCmd2, ',');
					sCmd2:= CONCAT(sCmd2, Payload_Rear);
					sCmd2:= CONCAT(sCmd2, ',');
					sCmd2:= CONCAT(sCmd2, Overload_Lead);
					sCmd2:= CONCAT(sCmd2, ',');
					sCmd2:= CONCAT(sCmd2, Overload_Rear);
					sCmd2:= CONCAT(sCmd2, ',');
					sCmd2:= CONCAT(sCmd2, Pressure_Lead); 
					sCmd2:= CONCAT(sCmd2, ',');
					sCmd2:= CONCAT(sCmd2, Pressure_Rear); 
					sCmd2:= CONCAT(sCmd2, ',');
					sCmd2:= CONCAT(sCmd2, Overpressure_Lead); 
					sCmd2:= CONCAT(sCmd2, ',');
					sCmd2:= CONCAT(sCmd2, Overpressure_Rear); 
					sCmd2:= CONCAT(sCmd2, ',');
					sCmd2:= CONCAT(sCmd2, EventCode);
					sCmd2:= CONCAT(sCmd2, ')');
					CONCAT2(ADR(sCmd), ADR(sCmd2), ADR(sCmd), SIZEOF(sCmd));
					
					IF fbSQLCommand.Execute(ADR(sCmd), SIZEOF(sCmd)) THEN
						IF fbSQLCommand.bError THEN
							nState := 255; 
						ELSE
							nState := nState+1; 
							pSec := Background_Time.cSec;
							
						END_IF
					END_IF
					
				4: 
					Counter := Counter + 1;
					Done	:= TRUE;
						
				255:
					nState := 0;
					
			END_CASE
			
		END_IF
	END_IF
END_IF

(*
(* save data to buffer every second *)
IF diff:= Background_Time.cSec <> pSec THEN

	IF Done THEN
		nState 	:= 0;
		Done	:= FALSE;	
	END_IF
	
	
	(* connect to localdb *)
	IF NOT fbSqlDatabase.bConnected THEN
		fbSqlDatabase.Connect(1);
	ELSE
	
		CASE nState OF
				
			0:
				IF fbSqlDatabase.CreateCmd(ADR(fbSqlCommand)) THEN
					IF fbSqlDatabase.bError THEN
						nState := 255; 
					ELSE
						nState := nState+1; 
					END_IF
				END_IF
				
			1:	
				(* build query *)	
				sCmd:= 'INSERT INTO buffer_data (datetime,trailer_id_lead,trailer_id_rear,latitude,longitude,speed,overspeed,payload_lead,payload_rear,overload_lead,overload_rear,pressure_lead,pressure_rear,overpressure_lead,overpressure_rear,event_code) VALUES ($'';
				sCmd2:= TimeStr;
				sCmd2:= CONCAT(sCmd2, '$',');
				sCmd2:= CONCAT(sCmd2, Trailer_ID_Lead);
				sCmd2:= CONCAT(sCmd2, ',');
				sCmd2:= CONCAT(sCmd2, Trailer_ID_Rear);
				sCmd2:= CONCAT(sCmd2, ',');
				sCmd2:= CONCAT(sCmd2, Lat);
				sCmd2:= CONCAT(sCmd2, ',');
				sCmd2:= CONCAT(sCmd2, Lon);
				sCmd2:= CONCAT(sCmd2, ',');
				sCmd2:= CONCAT(sCmd2, Speed);
				sCmd2:= CONCAT(sCmd2, ',');
				sCmd2:= CONCAT(sCmd2, Overspeed);
				sCmd2:= CONCAT(sCmd2, ',');
				sCmd2:= CONCAT(sCmd2, Payload_Lead);
				sCmd2:= CONCAT(sCmd2, ',');
				sCmd2:= CONCAT(sCmd2, Payload_Rear);
				sCmd2:= CONCAT(sCmd2, ',');
				sCmd2:= CONCAT(sCmd2, Overload_Lead);
				sCmd2:= CONCAT(sCmd2, ',');
				sCmd2:= CONCAT(sCmd2, Overload_Rear);
				sCmd2:= CONCAT(sCmd2, ',');
				sCmd2:= CONCAT(sCmd2, Pressure_Lead); 
				sCmd2:= CONCAT(sCmd2, ',');
				sCmd2:= CONCAT(sCmd2, Pressure_Rear); 
				sCmd2:= CONCAT(sCmd2, ',');
				sCmd2:= CONCAT(sCmd2, Overpressure_Lead); 
				sCmd2:= CONCAT(sCmd2, ',');
				sCmd2:= CONCAT(sCmd2, Overpressure_Rear); 
				sCmd2:= CONCAT(sCmd2, ',');
				sCmd2:= CONCAT(sCmd2, EventCode);
				sCmd2:= CONCAT(sCmd2, ')');
				CONCAT2(ADR(sCmd), ADR(sCmd2), ADR(sCmd), SIZEOF(sCmd));
				
				IF fbSQLCommand.Execute(ADR(sCmd), SIZEOF(sCmd)) THEN
					IF fbSQLCommand.bError THEN
						nState := 255; 
					ELSE
						nState := nState+1; 
						pSec := Background_Time.cSec;
						
					END_IF
				END_IF
				
			2: 
				Done		:= TRUE;	
				
			255:
				nState := 0;
	
		END_CASE
	END_IF
END_IF
*)

END_PROGRAM

// ---- POUs/Read_Payload.TcPOU
PROGRAM Read_Payload
VAR
	EL3061_Lead_Bit AT %I* 	: INT;
	EL3061_Rear_Bit AT %I* 	: INT;
	
	//axle of lead trailer
	R3_Bit			: REAL;
	R3_BitTare		: REAL := 8043;
	R31_BitPerTon	: REAL := 7.8864; //bit caused by payload on lead trailer
	R32_BitPerTon	: REAL := 7.8864; //bit caused by payload on rear trailer
	
	//axle of rear trailer
	R4_Bit			: REAL;
	R4_BitTare		: REAL := 8043;
	R42_BitPerTon	: REAL := 7.8864;
	
	Payload_Lead	: REAL;
	Payload_Rear	: REAL;
	Payload_Total	: REAL;	
	
	Threshold_Lead	: REAL := 40.5;
	Threshold_Rear	: REAL := 72;	
	Overload_Lead	: BOOL := FALSE;
	Overload_Rear	: BOOL := FALSE;
END_VAR

R3_Bit := INT_TO_REAL(EL3061_Lead_Bit);
R4_Bit := INT_TO_REAL(EL3061_Rear_Bit);

Payload_Rear	:= (R4_Bit - R4_BitTare) / R42_BitPerTon;
Payload_Lead	:= (R3_Bit - (R32_BitPerTon * Payload_Rear)) / R31_BitPerTon;
Payload_Total	:= Payload_Lead + Payload_Rear;

IF Payload_Lead < 0 THEN
	Payload_Lead := 0;
END_IF

IF Payload_Rear < 0 THEN
	Payload_Rear := 0;
END_IF

IF Payload_Lead > Threshold_Lead THEN
	Overload_Lead := TRUE;
ELSE
	Overload_Lead := FALSE;	
END_IF

IF Payload_Rear > Threshold_Rear THEN
	Overload_Rear := TRUE;
ELSE
	Overload_Rear := FALSE;	
END_IF

(*
IF Read_GPS.Speed < 1 AND Background_IMU.Pitch < 3 AND Background_IMU.Roll < 3 THEN
	Payload	:= Payload_Raw;
END_IF

(* check for overload *)
IF Payload > Threshold THEN
	Overload := TRUE;
ELSE
	Overload := FALSE;	
END_IF
*)

END_PROGRAM

// ---- POUs/Read_Pressure.TcPOU
PROGRAM Read_Pressure
VAR
	Pressure_Val	: REAL := 0;
	Pressure_Cyl	: REAL := 0;
	
	Hyd_Efficiency	: REAL := 0;
	nBit_Val AT %I*	: UINT;
	nBit_Cyl AT %I*	: UINT;
END_VAR

(* convert to pressure *)
Pressure_Val := (nBit_Val/32767)*160;
Pressure_Cyl := (nBit_Cyl/32767)*160;

(* calculate hyd efficiency *)
//rHyd_Efficiency := Read_Pressure.Pressure_Cyl / Read_Pressure.Pressure_Val;

END_PROGRAM

// ---- POUs/Main_Read.TcPOU
PROGRAM Main_Read
VAR
	TimeStr	: STRING;
END_VAR

(* get timestamp *)
TimeStr	:= Background_Time.TimeStr;

(* read sensors *)
Read_IMU();
Read_FatigueCam();
Read_GPS();
Read_Payload();
Read_Pressure();

END_PROGRAM

// ---- POUs/Read_FatigueCam.TcPOU
PROGRAM Read_FatigueCam
VAR
	fb_Receive		: FB_FatigueCam_Receive;
	fbSend			: SendData;
	bSendBusy		: BOOL;
	eSendErrorID	: ComError_t;
	nSendCounter	: UDINT;
	
	pSec	: WORD := 0;
	
	TimeStr		: STRING;
	Year		: USINT;
	Month		: USINT;
	bDate		: USINT;
	Hour		: USINT;
	Minute		: USINT;
	Second		: USINT;
	
	YearBin		: STRING;
	MonthBin	: STRING;
	bDateBin	: STRING;
	HourBin		: STRING;
	MinuteBin	: STRING;
	SecondBin	: STRING;
	
	BinStr		: ARRAY [1..4] OF STRING;
	TimeBin		: STRING;
	
	Synced		: BOOL;
	
	Command			: ULINT := 16#00;
	Sent_Command	: ULINT;
	Command_Sent	: BOOL;
	Response		: STRING := 'ABC';
	Prev_Response	: STRING;
	Response_Count	: INT;
	EventID			: STRING := '00';
	prevEventID		: STRING;
	EventCode		: STRING := '0';
	New_Event		: BOOL;
	
	Prefix		: WORD;
	LenPrefix	: BYTE;
	
	i	: INT;
END_VAR

(* receive response *)
Prefix		:= 16#AA;
LenPrefix	:= 1;	

(*
fb_Receive(
	RxBuffer	:= Background_FatigueCam.RxBuffer,
	Command		:= Command,
	Prefix		:= Prefix,
	LenPrefix	:= LenPrefix,
	EventID		=> EventID,
	EventCode	=> EventCode,
	Response	=> Response,
);
*)


IF Background_Time.cSec <> pSec THEN
	
	(* sync time every 1 minute *)
	(*
	IF pSec = 0 THEN 
		Synced := FALSE;
	END_IF
	
	IF Synced = FALSE THEN
		
		IF NOT Command_Sent AND Response <> LWORD_TO_HEXSTR(in := Sent_Command, iPrecision := 1, bLoCase := FALSE) THEN
			(* send sync command *)
			TimeStr		:= Background_Time.TimeStr; //get datetime
	
			Year		:= STRING_TO_USINT(MID(STR := TimeStr, LEN := 2, POS := 3));
			Month		:= STRING_TO_USINT(MID(STR := TimeStr, LEN := 2, POS := 6));
			bDate		:= STRING_TO_USINT(MID(STR := TimeStr, LEN := 2, POS := 9));
			Hour		:= STRING_TO_USINT(MID(STR := TimeStr, LEN := 2, POS := 12));
			Minute		:= STRING_TO_USINT(MID(STR := TimeStr, LEN := 2, POS := 15));
			Second		:= STRING_TO_USINT(MID(STR := TimeStr, LEN := 2, POS := 18));
			
			(* convert datetime to binary *)
			YearBin		:= BYTE_TO_BINSTR(in := Year, iPrecision := 6);
			MonthBin	:= BYTE_TO_BINSTR(in := Month, iPrecision := 4);
			bDateBin	:= BYTE_TO_BINSTR(in := bDate, iPrecision := 5);
			HourBin		:= BYTE_TO_BINSTR(in := Hour, iPrecision := 5);
			MinuteBin	:= BYTE_TO_BINSTR(in := Minute, iPrecision := 6);
			SecondBin	:= BYTE_TO_BINSTR(in := Second, iPrecision := 6);
			BinStr[4]	:= CONCAT(YearBin, MonthBin); 
			BinStr[4]	:= CONCAT(BinStr[4], bDateBin);
			BinStr[4]	:= CONCAT(BinStr[4], HourBin); 
			BinStr[4]	:= CONCAT(BinStr[4], MinuteBin);
			BinStr[4]	:= CONCAT(BinStr[4], SecondBin);
			
			(* separate bytes *)
			BinStr[1]	:= LEFT(STR := BinStr[4], SIZE := 8);
			BinStr[2]	:= MID(STR := BinStr[4], LEN := 8, POS := 9);
			BinStr[3]	:= MID(STR := BinStr[4], LEN := 8, POS := 17);
			BinStr[4]	:= RIGHT(STR := BinStr[4], SIZE := 8);
			
			(* build sync command *)
			TimeBin		:= CONCAT('2#', BinStr[4]);
			TimeBin		:= CONCAT(TimeBin, BinStr[3]);
			TimeBin		:= CONCAT(TimeBin, BinStr[2]);
			TimeBin		:= CONCAT(TimeBin, BinStr[1]);
			TimeBin		:= CONCAT(TimeBin, '10001101'); //8D
			TimeBin		:= CONCAT(TimeBin, '10101010'); //AA
			Command		:= STRING_TO_ULINT(TimeBin);
			
			Prefix := 16#8DAA;
			LenPrefix := 2;
			
			(* send command *)
			fbSend( 
				pSendData	:= ADR(Command),
				TXbuffer 	:= Background_FatigueCam.TxBuffer,
				Length 		:= SIZEOF(Command),
				Busy		=> bSendBusy,
				Error		=> 
			);
			IF fbSend.Error <> COMERROR_NOERROR THEN
				eSendErrorID := fbSend.Error;
			ELSE
				Command_Sent 	:= TRUE;
				Sent_Command 	:= Command;
				Response_Count	:= 0;
			END_IF

		ELSE
			Synced	:= TRUE;
			
		END_IF
		
		IF Command_Sent THEN
			(* receive response *)
			fb_Receive(
				RxBuffer	:= Background_FatigueCam.RxBuffer,
				Command		:= Command,
				Prefix		:= Prefix,
				LenPrefix	:= LenPrefix,
				EventID		=> EventID,
				EventCode	=> EventCode,
				Response	=> Response,
			);
			
			Response_Count := Response_Count + 1;
			
			IF Response <> Prev_Response THEN
				Prev_Response := Response;
				Command_Sent := FALSE;
			ELSIF Response_Count > 10 THEN
				Command_Sent := FALSE;			
			END_IF
		END_IF
		
		pSec 	:= Background_Time.cSec;
		
	ELSE
		(* fatigue cam request event *)
		Command		:= 16#000000008CAA;
		Prefix		:= 16#AA;
		LenPrefix	:= 1;	
		
		(* send command *)
		fbSend( 
			pSendData	:= ADR(Command),
			TXbuffer 	:= Background_FatigueCam.TxBuffer,
			Length 		:= SIZEOF(Command),
			Busy		=> bSendBusy,
			Error		=> 
		);
		IF fbSend.Error <> COMERROR_NOERROR THEN
			eSendErrorID := fbSend.Error;
		END_IF
		
		(* receive response *)
		fb_Receive(
			RxBuffer	:= Background_FatigueCam.RxBuffer,
			Command		:= Command,
			Prefix		:= Prefix,
			LenPrefix	:= LenPrefix,
			EventID		=> EventID,
			EventCode	=> EventCode,
			Response	=> Response,
		);
	
		pSec := Background_Time.cSec;
	
	END_IF
	*)
	
	IF EventCode = '' OR EventID = prevEventID THEN
		EventCode 	:= '0';
		i			:= 0;		
	ELSE
		i := i+1;
		IF i > 1 THEN
			prevEventID	:= EventID;
		END_IF		
	END_IF
	
	pSec := Background_Time.cSec;
	
END_IF

END_PROGRAM

// ---- POUs/Background_FatigueCam.TcPOU
PROGRAM Background_FatigueCam
VAR
	(* ----------------- via db9 -------------------*)	
	(* I/O variables for a PC-COM port *)
    stIn_PcCom AT %I* : PcComInData; (* linked to the port in the TwinCAT System Manager *)
    stOut_PcCom AT %Q* : PcComOutData; (* linked to the port in the TwinCAT System Manager *)
    RxBuffer     : ComBuffer; (* Receive data buffer; used with all receive function blocks *)
    TxBuffer     : ComBuffer; (* Transmit data buffer; used with all receive function blocks *)
	
	(* background communication with the PC COM port device *)
    fbPcComCtrl       : SerialLineControl;
    bPcComCtrlError   : BOOL;
    ePcComCtrlErrorID : ComError_t;
	
	(* ----------------- via el6001 -------------------*)
	(* background communication with the EL6001 terminal *)
	(*
	RxBuffer	:ComBuffer;
	TxBuffer	:ComBuffer;
	
	fbEL6001Ctrl		: SerialLineControl;
	bEL6001CtrlError	: BOOL;
	eEL6001CtrlErrorID	: ComError_t;
	(* 	I/O variables for a EL6001 terminal*)
	stIn_EL6001 AT %I*	: EL6inData22B;	(* linked to the EL6001 in the TwinCAT System Manager *)
	stOut_EL6001 AT %Q*	: EL6outData22B;(* linked to the EL6001 in the TwinCAT System Manager *)
	*)
END_VAR

(* ---------------------- via db9 ------------------ *)
(* background communication with the PC COM port device *)
fbPcComCtrl(
    Mode      := SERIALLINEMODE_PC_COM_PORT, 
    pComIn    := ADR(stIn_PcCom), 
    pComOut   := ADR(stOut_PcCom), 
    SizeComIn := SIZEOF(stIn_PcCom), 
    Error     => bPcComCtrlError, 
    ErrorID   => ePcComCtrlErrorID, 
    TxBuffer  := TxBuffer, 
    RxBuffer  := RxBuffer 
);

(* ---------------------- via el6001 ------------------ *)
(*
(*
The SerialLineControl function block is supposed to be called in every PLC cycle.
It communicates with the serial line hardware device and transmits or receives data.
The SerialLineControl can be called in the standard task (e.g.for PcCOM port usage) 
or in a separate fast task (e.g.for terminal usage) as well.
A fast separate task will be necessary at high baud rates or with KL6001 terminals 
which have a small process image (3 or 5 data bytes only)
*)

(* background communication with the EL6001 terminal *)
fbEL6001Ctrl(
	Mode:= SERIALLINEMODE_EL6_22B, 
	pComIn:= ADR(stIn_EL6001), 
	pComOut:= ADR(stOut_EL6001), 
	SizeComIn:= SIZEOF(stIn_EL6001), 
	Error=> , 
	ErrorID=> , 
	TxBuffer:= TxBuffer, 
	RxBuffer:= RxBuffer );
IF fbEL6001Ctrl.Error THEN
	bEL6001CtrlError := TRUE;
	eEL6001CtrlErrorID := fbEL6001Ctrl.ErrorID;
END_IF
*)

END_PROGRAM

// ---- POUs/Read_GPS.TcPOU
PROGRAM Read_GPS
VAR
	(* receive string variables *)
	fbReceiveString	: ReceiveString;
	DataString		: STRING;
	Pref			: STRING := '$$GPRMC,';
	Suff			: STRING := '*';
	
	(* parsing variables *)
    sSeparator   : STRING(1) := ',';
	sSeparator2  : STRING(1) := '.';
    aSplit       : ARRAY[1..cMax] OF STRING; //parsed string
    bResultSplit : BOOL;
    i            : UDINT;
	
	(* gps variables *)
	HourInt		: INT;
	HourStr		: STRING;
	TimeStamp	: STRING;
	LatLeftStr	: STRING;
	LatRightStr	: STRING;
	LonLeftStr	: STRING;
	LonRightStr	: STRING;
	LatLeft		: INT;
	LatRight	: INT;
	LonLeft		: INT;
	LonRight	: INT;
	LatDeg		: REAL;
	LonDeg		: REAL;
	LatMin		: REAL;
	LonMin		: REAL;
	Lat			: REAL;
	Lon			: REAL;
	Speed		: REAL;
	Threshold	: REAL := 60;
	Overspeed	: BOOL := FALSE;
	
	Cycle_Duration	: STRING := '0';
	
	pSec	: WORD;
END_VAR

VAR CONSTANT
    cMax         : UDINT := 11; //no. of substrings
END_VAR

IF Background_Time.cSec <> pSec THEN

	(* get gps data string *)
	fbReceiveString(
		RxBuffer := Background_GPS.RxBuffer, 
		Prefix := Pref, 
		Suffix := Suff, 
		Timeout := T#1S, 
		ReceivedString := DataString
	);
	
	(* gps data parsing *)
	aSplit[1] := DataString;
	FOR i:=1 TO cMax-1 DO
		bResultSplit := FindAndSplit( 
							pSeparator     := ADR(sSeparator),  
							pSrcString := ADR(aSplit[i]), 
							pLeftString    := ADR(aSplit[i]),   
							nLeftSize  := SIZEOF(aSplit[i]), 
							pRightString   := ADR(aSplit[i+1]), 
							nRightSize := SIZEOF(aSplit[i+1]),
							bSearchFromRight := FALSE 
						);
		IF NOT bResultSplit THEN
			EXIT;
		END_IF
	END_FOR
	
	IF aSplit[3] = 'A' THEN
		(* latitude & longitude conversion *)
		FindAndSplit( 
			pSeparator     		:= ADR(sSeparator2),  
			pSrcString 			:= ADR(aSplit[4]), 
			pLeftString    		:= ADR(LatLeftStr),   
			nLeftSize  			:= SIZEOF(LatLeftStr), 
			pRightString   		:= ADR(LatRightStr), 
			nRightSize 			:= SIZEOF(LatRightStr),
			bSearchFromRight 	:= FALSE 
		);
		
		FindAndSplit( 
			pSeparator     		:= ADR(sSeparator2),  
			pSrcString 			:= ADR(aSplit[6]), 
			pLeftString    		:= ADR(LonLeftStr),   
			nLeftSize  			:= SIZEOF(LonLeftStr), 
			pRightString   		:= ADR(LonRightStr), 
			nRightSize 			:= SIZEOF(LonRightStr),
			bSearchFromRight 	:= FALSE 
		);
		
		LatLeft 	:= STRING_TO_INT(LatLeftStr);
		LatRight 	:= STRING_TO_INT(LatRightStr);
		LonLeft 	:= STRING_TO_INT(LonLeftStr);
		LonRight 	:= STRING_TO_INT(LonRightStr);
		Lat			:= INT_TO_REAL(LatLeft) + (INT_TO_REAL(LatRight)/EXPT(10,LEN(LatRightStr)));
		Lon 		:= INT_TO_REAL(LonLeft) + (INT_TO_REAL(LonRight)/EXPT(10,LEN(LonRightStr)));;
		LatDeg 		:= TRUNC(Lat/100);
		LonDeg 		:= TRUNC(Lon/100);
		LatMin 		:= Lat - (LatDeg*100);
		LonMin 		:= Lon - (LonDeg*100);
		Lat 		:= LatDeg + (LatMin/60);
		Lon			:= LonDeg + (LonMin/60);
		
		IF aSplit[5] = 'S' THEN
			Lat := Lat*(-1);
		END_IF
		
		IF aSplit[7] = 'W' THEN
			Lon := Lon*(-1); 
		END_IF
		
		(* speed conversion *)
		Speed	:= STRING_TO_REAL(aSplit[8]) * 1.852;
		
		(* check for overspeed *)
		IF Speed > Threshold THEN
			Overspeed := TRUE;
		ELSE
			Overspeed := FALSE;
		END_IF
		
		(* calculate cycle time *)
		//Cycle_Duration :=
	ELSE
		(* gps no signal error handling *)
	END_IF
	
	pSec := Background_Time.cSec;
	
END_IF

END_PROGRAM

// ---- POUs/Vacuum_Buffer_Data.TcPOU
PROGRAM Vacuum_Buffer_Data
VAR
	fbSqlDatabase	: FB_SQLDatabaseEvt(sNetID := '', tTimeout := T#1000S);
	fbSqlCommand	: FB_SQLCommandEvt(sNetID := '', tTimeout := T#1000S);
	fbSqlResult		: FB_SQLResultEvt(sNetID :='', tTimeout   := T#1000S); 
	nState			: INT;
	sCmd			: STRING(500000);
	Vacuumed		: BOOL;
END_VAR

CASE nState OF
				
		0:
			(* connect to buffer_imu *)		
			IF fbSqlDatabase.Connect(1) THEN
				IF fbSqlDatabase.bError THEN
					nState := 255; 
				ELSE
					IF fbSqlDatabase.bConnected THEN
						nState := nState+1;
					END_IF 
				END_IF
			END_IF
			
		1:
			IF fbSqlDatabase.CreateCmd(ADR(fbSqlCommand)) THEN
				IF fbSqlDatabase.bError THEN
					nState := 255; 
				ELSE
					nState := nState+1; 
				END_IF
			END_IF
		
		2:	
			IF NOT Vacuumed THEN
				(* build query *)	
				sCmd	:= 'VACUUM';
				
				IF fbSQLCommand.Execute(ADR(sCmd), SIZEOF(sCmd)) THEN
					IF fbSQLCommand.bError THEN
						nState := 255; 
					ELSE
						nState 		:= nState+1; 
					END_IF
				END_IF
				
			ELSE 
				nState := nState+1;
			END_IF
		
		3:
			IF fbSqlDatabase.Disconnect() THEN
				IF fbSqlDatabase.bError THEN
					nState := 255;
				ELSE
					nState 		:= nState+1;
					Vacuumed 	:= TRUE;
				END_IF
			END_IF
			
		255:
			nState := 0;
			
END_CASE

END_PROGRAM

// ---- POUs/Send_Data.TcPOU
PROGRAM Send_Data
VAR
	fbMqttClient : FB_IotMqttClient;
	bSetParameter : BOOL := TRUE;
	bConnect : BOOL := TRUE;
	
	(* aws certificates *)
	
	(*------------------ actual ----------------*)
	(*
	rootCA		: STRING(255) := 'C:\Users\Administrator\Downloads\AWSCert\AmazonRootCA1.pem';
	thingCert	: STRING(255) := 'C:\Users\Administrator\Downloads\AWSCert\a2ca8bd1ed97a43e38f2bffcdf7ca64a29d3483826fdb03b3eb616af8a5efc9e-certificate.pem.crt';
	privateKey	: STRING(255) := 'C:\Users\Administrator\Downloads\AWSCert\a2ca8bd1ed97a43e38f2bffcdf7ca64a29d3483826fdb03b3eb616af8a5efc9e-private.pem.key';
	*)
	
	rootCA		: STRING(255) := 'C:\Users\Administrator\Downloads\AWSCert\AmazonRootCA1.pem';
	thingCert	: STRING(255) := 'C:\Users\Administrator\Downloads\AWSCert\8872c9f9d2c9335079f20c0506a3dd3599fd4d8552622bd2d7f8ae6d1681c64f-certificate.pem.crt';
	privateKey	: STRING(255) := 'C:\Users\Administrator\Downloads\AWSCert\8872c9f9d2c9335079f20c0506a3dd3599fd4d8552622bd2d7f8ae6d1681c64f-private.pem.key';
	
	(* ------------------ test ------------------ *)
	(*
	rootCA		: STRING(255) := 'C:\Users\muhammad.rahman\Downloads\double-sdt-1-certs\AmazonRootCA1.pem';
	thingCert	: STRING(255) := 'C:\Users\muhammad.rahman\Downloads\double-sdt-test-certs\8872c9f9d2c9335079f20c0506a3dd3599fd4d8552622bd2d7f8ae6d1681c64f-certificate.pem.crt';
	privateKey	: STRING(255) := 'C:\Users\muhammad.rahman\Downloads\double-sdt-test-certs\8872c9f9d2c9335079f20c0506a3dd3599fd4d8552622bd2d7f8ae6d1681c64f-private.pem.key';
	*)
	
	(* broker settings *)
	endpoint	: STRING := 'a2o01t3xth0mr1-ats.iot.ap-southeast-1.amazonaws.com';
	port		: UINT := 8883;
	//clientID	: STRING := 'double-sdt-1';
	clientID	: STRING := 'double-sdt-test';
	
	(* published message *)
	sTopicPub 	: STRING(255) := 'iot/smartproduct/mifa/double-sdt/data'; //message topic
	sPayloadPub 	: STRING(500000);
	str				: STRING(100000);
	valSeparator	: STRING := '","';
	comma			: STRING := ',';
	arrayEnd		: STRING := '"]';
	arrayEnd2		: STRING := ']';
	msgEnd			: STRING := '}';
	i				: ULINT;
	
	(* topic subscription *)
	bSubscribed : BOOL;
	sTopicSub 	: STRING(255) := 'iot/smartproduct/mifa/double-sdt/data';
	
	(* received message *)	
	{attribute 'TcEncoding':='UTF-8'}
	sTopicRcv : STRING(255);
	{attribute 'TcEncoding':='UTF-8'}
	sPayloadRcv : STRING(255);
	
	fbMessageQueue : FB_IotMqttMessageQueue;
	fbMessage : FB_IotMqttMessage;
	
	hrErrorOccurred : HRESULT; // contains the latest occurred error
	Published		: BOOL;
	Publish			: BOOL;
END_VAR

IF Main_SendData.New_Data THEN
	Publish		:= FALSE;
	Published 	:= FALSE;	
END_IF


IF bSetParameter THEN
	bSetParameter := FALSE;
	
	(* TLS settings for AWS IoT connection *)
	fbMqttClient.stTLS.sCA 		:= rootCA; //root CA
    fbMqttClient.stTLS.sCert 	:= thingCert; //certificate of thing
    fbMqttClient.stTLS.sKeyFile := privateKey; //private key of thing
	
	(* Broker settings für AWS IoT *)
	fbMqttClient.sHostName:= endpoint; //broker endpoint
	fbMqttClient.nHostPort:= port; //default mqtt tls port
	fbMqttClient.sClientId:= clientID; //client id
	fbMqttClient.sTopicPrefix:= ''; 
	
	fbMqttClient.ipMessageQueue := fbMessageQueue;
END_IF

(* connect to mqtt broker *)
fbMqttClient.Execute(bConnect); 
IF fbMqttClient.bError THEN
	// add your error logging here
	hrErrorOccurred := fbMqttClient.hrErrorCode;
END_IF

IF fbMqttClient.bConnected THEN	
	IF NOT bSubscribed THEN
		bSubscribed := fbMqttClient.Subscribe(sTopic:=sTopicSub, eQoS:=TcIotMqttQos.AtMostOnceDelivery); //subscribe to topic
		IF fbMqttClient.bError THEN
			// add your error logging here
			hrErrorOccurred := fbMqttClient.hrErrorCode;
		END_IF
	END_IF
	
	(* build message payload *)
	sPayloadPub := CONCAT('{"primemover_id":', Read_ID.PrimeMover_ID);
	
	(* lead trailer id string *)
	str	:= ',"trailer_id_lead":[';
	FOR i:=1 TO Get_Data.Data_Length BY 1 DO
		CONCAT2(ADR(str), ADR(Get_Data.Trailer_ID_Lead[i]), ADR(str), SIZEOF(str)); 
		
		IF i <> Get_Data.Data_Length THEN
			CONCAT2(ADR(str), ADR(comma), ADR(str), SIZEOF(str));
		ELSE
			CONCAT2(ADR(str), ADR(arrayEnd2), ADR(str), SIZEOF(str));
		END_IF
		
	END_FOR
	
	CONCAT2(ADR(sPayloadPub), ADR(str), ADR(sPayloadPub), SIZEOF(sPayloadPub));
	
	(* rear trailer id string *)
	str	:= ',"trailer_id_rear":[';
	FOR i:=1 TO Get_Data.Data_Length BY 1 DO
		CONCAT2(ADR(str), ADR(Get_Data.Trailer_ID_Rear[i]), ADR(str), SIZEOF(str)); 
		
		IF i <> Get_Data.Data_Length THEN
			CONCAT2(ADR(str), ADR(comma), ADR(str), SIZEOF(str));
		ELSE
			CONCAT2(ADR(str), ADR(arrayEnd2), ADR(str), SIZEOF(str));
		END_IF
		
	END_FOR
	
	CONCAT2(ADR(sPayloadPub), ADR(str), ADR(sPayloadPub), SIZEOF(sPayloadPub));
	
	(* date time string *)
	str	:= ',"datetime":["';
	FOR i:=1 TO Get_Data.Data_Length BY 1 DO
		CONCAT2(ADR(str), ADR(Get_Data.TimeStr[i]), ADR(str), SIZEOF(str)); 
		
		IF i <> Get_Data.Data_Length THEN
			CONCAT2(ADR(str), ADR(valSeparator), ADR(str), SIZEOF(str));
		ELSE
			CONCAT2(ADR(str), ADR(arrayEnd), ADR(str), SIZEOF(str));
		END_IF
		
	END_FOR
	
	CONCAT2(ADR(sPayloadPub), ADR(str), ADR(sPayloadPub), SIZEOF(sPayloadPub));
	
	(* latitude string *)
	str	:= ',"latitude":[';
	FOR i:=1 TO Get_Data.Data_Length BY 1 DO
		CONCAT2(ADR(str), ADR(Get_Data.Lat[i]), ADR(str), SIZEOF(str)); 
		
		IF i <> Get_Data.Data_Length THEN
			CONCAT2(ADR(str), ADR(comma), ADR(str), SIZEOF(str));
		ELSE
			CONCAT2(ADR(str), ADR(arrayEnd2), ADR(str), SIZEOF(str));
		END_IF
		
	END_FOR
	
	CONCAT2(ADR(sPayloadPub), ADR(str), ADR(sPayloadPub), SIZEOF(sPayloadPub));
	
	(* longitude string *)
	str	:= ',"longitude":[';
	FOR i:=1 TO Get_Data.Data_Length BY 1 DO
		CONCAT2(ADR(str), ADR(Get_Data.Lon[i]), ADR(str), SIZEOF(str)); 
		
		IF i <> Get_Data.Data_Length THEN
			CONCAT2(ADR(str), ADR(comma), ADR(str), SIZEOF(str));
		ELSE
			CONCAT2(ADR(str), ADR(arrayEnd2), ADR(str), SIZEOF(str));
		END_IF
		
	END_FOR
	
	CONCAT2(ADR(sPayloadPub), ADR(str), ADR(sPayloadPub), SIZEOF(sPayloadPub));
	
	(* speed string *)
	str	:= ',"speed":[';
	FOR i:=1 TO Get_Data.Data_Length BY 1 DO
		CONCAT2(ADR(str), ADR(Get_Data.Speed[i]), ADR(str), SIZEOF(str)); 
		
		IF i <> Get_Data.Data_Length THEN
			CONCAT2(ADR(str), ADR(comma), ADR(str), SIZEOF(str));
		ELSE
			CONCAT2(ADR(str), ADR(arrayEnd2), ADR(str), SIZEOF(str));
		END_IF
		
	END_FOR
	
	CONCAT2(ADR(sPayloadPub), ADR(str), ADR(sPayloadPub), SIZEOF(sPayloadPub));
	
	(* overspeed string *)
	str	:= ',"overspeed":[';
	FOR i:=1 TO Get_Data.Data_Length BY 1 DO
		CONCAT2(ADR(str), ADR(Get_Data.Overspeed[i]), ADR(str), SIZEOF(str)); 
		
		IF i <> Get_Data.Data_Length THEN
			CONCAT2(ADR(str), ADR(comma), ADR(str), SIZEOF(str));
		ELSE
			CONCAT2(ADR(str), ADR(arrayEnd2), ADR(str), SIZEOF(str));
		END_IF
		
	END_FOR
	
	CONCAT2(ADR(sPayloadPub), ADR(str), ADR(sPayloadPub), SIZEOF(sPayloadPub));
	
	(* payload lead string *)
	str	:= ',"payload_lead":[';
	FOR i:=1 TO Get_Data.Data_Length BY 1 DO
		CONCAT2(ADR(str), ADR(Get_Data.Payload_Lead[i]), ADR(str), SIZEOF(str)); 
		
		IF i <> Get_Data.Data_Length THEN
			CONCAT2(ADR(str), ADR(comma), ADR(str), SIZEOF(str));
		ELSE
			CONCAT2(ADR(str), ADR(arrayEnd2), ADR(str), SIZEOF(str));
		END_IF
		
	END_FOR
	
	CONCAT2(ADR(sPayloadPub), ADR(str), ADR(sPayloadPub), SIZEOF(sPayloadPub));
	
